    //---------------------------------------------------------------------
    // 6. RESET CHANNEL STATUS
    //---------------------------------------------------------------------
    ChannelStatus.Enable := FALSE;
    ChannelStatus.Online := FALSE;
    ChannelStatus.Ready := FALSE;
    ChannelStatus.Busy := FALSE;
    ChannelStatus.ResultReady := FALSE;
    ChannelStatus.Error := FALSE;
    ChannelStatus.CurrentJobID := 0;
    ChannelStatus.CurrentTriggerID := 0;
    ChannelStatus.ResultStatus := E_VisionResultStatus.VIS_RESULT_NONE;

    tHeartbeatTimeout(IN := FALSE);

    RETURN;
END_IF;


//=============================================================================
// DISABLE
//=============================================================================
IF NOT Enable THEN

    Registers[uiR2V + 0] := WORD#0;

    Active := FALSE;
    Error := FALSE;
    ErrorID := 0;

    ChannelStatus.Enable := FALSE;
    ChannelStatus.Online := FALSE;
    ChannelStatus.Ready := FALSE;
    ChannelStatus.Busy := FALSE;
    ChannelStatus.ResultReady := FALSE;
    ChannelStatus.Error := FALSE;

    RETURN;
END_IF;


//=============================================================================
// NORMAL RUN
//=============================================================================
Active := TRUE;
ChannelStatus.Enable := TRUE;

// Active := TRUE;
// ChannelStatus.Enable := TRUE;

// //=============================================================================
// // MEMORY BASE / SCALE
// //=============================================================================
// uiBase := Config.BaseAddress;
// uiR2V := uiBase + Config.CommandOffset;
// uiV2R := uiBase + Config.StatusOffset;
// uiData := uiBase + Config.DataOffset;
// uiMulti := uiBase + 132;                            // MultiData cố định theo mapping V1.1.
// 
// IF uiR2V + 99 > 1199 OR uiV2R + 199 > 1199 THEN
//     Error := TRUE;
//     ErrorID := 9251;                                // Base/Offset vượt vùng MODBUS.
//     RETURN;
// END_IF;

Error := FALSE;
ErrorID := 0;
rPositionScale := Config.PositionScale;
rAngleScale := Config.AngleScale;
rScoreScale := Config.ScoreScale;
IF ABS(rPositionScale) <= GVL.C_EPSILON THEN rPositionScale := 1.0; END_IF;
IF ABS(rAngleScale) <= GVL.C_EPSILON THEN rAngleScale := 1.0; END_IF;
IF ABS(rScoreScale) <= GVL.C_EPSILON THEN rScoreScale := 1.0; END_IF;

//=============================================================================
// 1. ROBOT -> VISION: CONTROL WORD + COMMAND
//=============================================================================
// Heartbeat dùng biến nội bộ toggle; KHÔNG đảo trực tiếp register mỗi scan Communication.
xHeartbeatToggle := NOT xHeartbeatToggle;

wControl := WORD#0;
wControl.0 := xHeartbeatToggle;
wControl.1 := Command.Execute;
wControl.2 := ModbusControl.RunCalib;
wControl.3 := ModbusControl.CalibPosReady;
wControl.4 := ModbusControl.AckResult;
wControl.5 := ModbusControl.AckBlock;
wControl.6 := Command.Reset;
wControl.7 := Command.Abort;
Registers[uiR2V + 0] := wControl;
Registers[uiR2V + 1] := UINT_TO_WORD(Command.JobID);

CASE Command.Application OF
    E_VisionApplication.VIS_APP_ALIGN: Registers[uiR2V + 2] := WORD#10;
    E_VisionApplication.VIS_APP_INSPECTION: Registers[uiR2V + 2] := WORD#20;
    E_VisionApplication.VIS_APP_SINGLE_POINT: Registers[uiR2V + 2] := WORD#30;
    E_VisionApplication.VIS_APP_POINT_LIST: Registers[uiR2V + 2] := WORD#40;
    E_VisionApplication.VIS_APP_GLUE_PATH: Registers[uiR2V + 2] := WORD#50;
    E_VisionApplication.VIS_APP_PICK_POSITION: Registers[uiR2V + 2] := WORD#60;
    E_VisionApplication.VIS_APP_CONVEYOR_PICK: Registers[uiR2V + 2] := WORD#70;
    E_VisionApplication.VIS_APP_CONVEYOR_INSPECTION: Registers[uiR2V + 2] := WORD#80;
    E_VisionApplication.VIS_APP_CONVEYOR_GLUE: Registers[uiR2V + 2] := WORD#90;
    E_VisionApplication.VIS_APP_CALIBRATION: Registers[uiR2V + 2] := WORD#100;
    ELSE Registers[uiR2V + 2] := WORD#0;
END_CASE;

Registers[uiR2V + 3] := F_VisionUDINTLowWord(Command.TriggerID);
Registers[uiR2V + 4] := F_VisionUDINTHighWord(Command.TriggerID);
Registers[uiR2V + 5] := UINT_TO_WORD(ModbusControl.CalibPointCount);
Registers[uiR2V + 6] := UINT_TO_WORD(ModbusControl.RequestBlockIndex);
Registers[uiR2V + 7] := UINT_TO_WORD(ModbusControl.AckBlockIndex);
Registers[uiR2V + 8] := UINT_TO_WORD(ModbusControl.CommandCode);
Registers[uiR2V + 9] := WORD#0;

// 12 Calibration Point; mỗi Point = X/Y/A, mỗi thành phần = LOW/HIGH WORD.
FOR uiPoint := 1 TO 12 DO
    diRaw := F_VisionRealToRawDINT(ModbusControl.CalibrationPoints[uiPoint].X, rPositionScale);
    Registers[uiR2V + 10 + (uiPoint - 1) * 6] := F_VisionDINTLowWord(diRaw);
    Registers[uiR2V + 11 + (uiPoint - 1) * 6] := F_VisionDINTHighWord(diRaw);

    diRaw := F_VisionRealToRawDINT(ModbusControl.CalibrationPoints[uiPoint].Y, rPositionScale);
    Registers[uiR2V + 12 + (uiPoint - 1) * 6] := F_VisionDINTLowWord(diRaw);
    Registers[uiR2V + 13 + (uiPoint - 1) * 6] := F_VisionDINTHighWord(diRaw);

    diRaw := F_VisionRealToRawDINT(ModbusControl.CalibrationPoints[uiPoint].A, rAngleScale);
    Registers[uiR2V + 14 + (uiPoint - 1) * 6] := F_VisionDINTLowWord(diRaw);
    Registers[uiR2V + 15 + (uiPoint - 1) * 6] := F_VisionDINTHighWord(diRaw);
END_FOR;

// Capture reference của command runtime.
diRaw := F_VisionRealToRawDINT(Command.CaptureConveyorPos, rPositionScale);
Registers[uiR2V + 82] := F_VisionDINTLowWord(diRaw);
Registers[uiR2V + 83] := F_VisionDINTHighWord(diRaw);

diRaw := F_VisionRealToRawDINT(Command.CaptureRobotPos.X, rPositionScale);
Registers[uiR2V + 84] := F_VisionDINTLowWord(diRaw);
Registers[uiR2V + 85] := F_VisionDINTHighWord(diRaw);

diRaw := F_VisionRealToRawDINT(Command.CaptureRobotPos.Y, rPositionScale);
Registers[uiR2V + 86] := F_VisionDINTLowWord(diRaw);
Registers[uiR2V + 87] := F_VisionDINTHighWord(diRaw);

diRaw := F_VisionRealToRawDINT(Command.CaptureRobotPos.A, rAngleScale);
Registers[uiR2V + 88] := F_VisionDINTLowWord(diRaw);
Registers[uiR2V + 89] := F_VisionDINTHighWord(diRaw);

//=============================================================================
// 2. VISION -> ROBOT: STATUS WORD
//=============================================================================
wStatus := Registers[uiV2R + 0];
ModbusStatus.HeartBeat := wStatus.0;
ModbusStatus.TriggerDone := wStatus.1;
ModbusStatus.CalibDone := wStatus.2;
ModbusStatus.ResultReady := wStatus.3;
ModbusStatus.Busy := wStatus.4;
ModbusStatus.Run1Slot := wStatus.5;
ModbusStatus.BlockReady := wStatus.6;
ModbusStatus.Error := wStatus.7;
ModbusStatus.CalibBusy := wStatus.8;
ModbusStatus.CalibError := wStatus.9;

ChannelStatus.Ready := NOT ModbusStatus.Busy AND NOT ModbusStatus.Error;
ChannelStatus.Busy := ModbusStatus.Busy;
ChannelStatus.ResultReady := ModbusStatus.ResultReady;
ChannelStatus.Error := ModbusStatus.Error;

// Heartbeat timeout 2 s: mỗi lần bit đổi thì reset timer.
IF ModbusStatus.HeartBeat <> xLastHeartbeat THEN
    xLastHeartbeat := ModbusStatus.HeartBeat;
    ChannelStatus.Online := TRUE;
    tHeartbeatTimeout(IN := FALSE);
ELSE
    tHeartbeatTimeout(IN := TRUE, PT := T#2S);
    IF tHeartbeatTimeout.Q THEN ChannelStatus.Online := FALSE; END_IF;
END_IF;

//=============================================================================
// 3. RESULT HEADER
//=============================================================================
ChannelStatus.CurrentJobID := WORD_TO_UINT(Registers[uiV2R + 1]);
udiTriggerID := F_VisionWordsToUDINT_LH(Registers[uiV2R + 4], Registers[uiV2R + 5]);
ChannelStatus.CurrentTriggerID := udiTriggerID;

VisionResult.Header.CameraID := Config.CameraID;
VisionResult.Header.JobID := WORD_TO_UINT(Registers[uiV2R + 1]);
VisionResult.Header.TriggerID := udiTriggerID;
VisionResult.Header.ResultCode := WORD_TO_UINT(Registers[uiV2R + 7]);
VisionResult.Header.ErrorCode := WORD_TO_UINT(Registers[uiV2R + 7]);
VisionResult.Header.DataCount := WORD_TO_UINT(Registers[uiV2R + 8]);
VisionResult.Header.BlockCount := WORD_TO_UINT(Registers[uiV2R + 9]);
VisionResult.Header.BlockIndex := WORD_TO_UINT(Registers[uiV2R + 10]);
VisionResult.Header.BlockDataCount := WORD_TO_UINT(Registers[uiV2R + 11]);
VisionResult.Header.Checksum := F_VisionWordsToUDINT_LH(Registers[uiV2R + 12], Registers[uiV2R + 13]);

diRaw := F_VisionWordsToDINT_LH(Registers[uiV2R + 14], Registers[uiV2R + 15]);
VisionResult.Header.CaptureConveyorPos := DINT_TO_REAL(diRaw) * rPositionScale;
ModbusStatus.BlockIndex := VisionResult.Header.BlockIndex;
ModbusStatus.BlockDataCount := VisionResult.Header.BlockDataCount;

CASE WORD_TO_UINT(Registers[uiV2R + 2]) OF
    10: VisionResult.Header.Application := E_VisionApplication.VIS_APP_ALIGN;
    20: VisionResult.Header.Application := E_VisionApplication.VIS_APP_INSPECTION;
    30: VisionResult.Header.Application := E_VisionApplication.VIS_APP_SINGLE_POINT;
    40: VisionResult.Header.Application := E_VisionApplication.VIS_APP_POINT_LIST;
    50: VisionResult.Header.Application := E_VisionApplication.VIS_APP_GLUE_PATH;
    60: VisionResult.Header.Application := E_VisionApplication.VIS_APP_PICK_POSITION;
    70: VisionResult.Header.Application := E_VisionApplication.VIS_APP_CONVEYOR_PICK;
    80: VisionResult.Header.Application := E_VisionApplication.VIS_APP_CONVEYOR_INSPECTION;
    90: VisionResult.Header.Application := E_VisionApplication.VIS_APP_CONVEYOR_GLUE;
    100: VisionResult.Header.Application := E_VisionApplication.VIS_APP_CALIBRATION;
    ELSE VisionResult.Header.Application := E_VisionApplication.VIS_APP_NONE;
END_CASE;

CASE WORD_TO_UINT(Registers[uiV2R + 3]) OF
    10: VisionResult.Header.DataType := E_VisionDataType.VIS_DATA_BOOL;
    20: VisionResult.Header.DataType := E_VisionDataType.VIS_DATA_VALUE;
    30: VisionResult.Header.DataType := E_VisionDataType.VIS_DATA_POS;
    40: VisionResult.Header.DataType := E_VisionDataType.VIS_DATA_ALIGN;
    50: VisionResult.Header.DataType := E_VisionDataType.VIS_DATA_INSPECTION;
    60: VisionResult.Header.DataType := E_VisionDataType.VIS_DATA_POINT_LIST;
    70: VisionResult.Header.DataType := E_VisionDataType.VIS_DATA_GLUE_PATH;
    80: VisionResult.Header.DataType := E_VisionDataType.VIS_DATA_TRACK_OBJECT;
    ELSE VisionResult.Header.DataType := E_VisionDataType.VIS_DATA_NONE;
END_CASE;

CASE WORD_TO_UINT(Registers[uiV2R + 6]) OF
    10: VisionResult.Header.ResultStatus := E_VisionResultStatus.VIS_RESULT_PENDING;
    20: VisionResult.Header.ResultStatus := E_VisionResultStatus.VIS_RESULT_OK;
    30: VisionResult.Header.ResultStatus := E_VisionResultStatus.VIS_RESULT_NG;
    40: VisionResult.Header.ResultStatus := E_VisionResultStatus.VIS_RESULT_NOT_FOUND;
    50: VisionResult.Header.ResultStatus := E_VisionResultStatus.VIS_RESULT_LOW_SCORE;
    60: VisionResult.Header.ResultStatus := E_VisionResultStatus.VIS_RESULT_OUT_OF_RANGE;
    70: VisionResult.Header.ResultStatus := E_VisionResultStatus.VIS_RESULT_INCOMPLETE;
    80: VisionResult.Header.ResultStatus := E_VisionResultStatus.VIS_RESULT_INVALID;
    900: VisionResult.Header.ResultStatus := E_VisionResultStatus.VIS_RESULT_ERROR;
    ELSE VisionResult.Header.ResultStatus := E_VisionResultStatus.VIS_RESULT_NONE;
END_CASE;
ChannelStatus.ResultStatus := VisionResult.Header.ResultStatus;

// Vision đã hạ ResultReady: kết thúc handshake Result trước.
IF NOT ModbusStatus.ResultReady THEN
    ModbusControl.AckResult := FALSE;
    ModbusControl.AckBlock := FALSE;
    ModbusControl.AckBlockIndex := 0;
    ModbusControl.RequestBlockIndex := 0;
END_IF;

//=============================================================================
// 4. SIMPLE RESULT - POS / ALIGN
//=============================================================================
IF ModbusStatus.ResultReady AND udiTriggerID <> 0 AND udiTriggerID <> udiLastResultTriggerID
AND (VisionResult.Header.DataType = E_VisionDataType.VIS_DATA_POS OR VisionResult.Header.DataType = E_VisionDataType.VIS_DATA_ALIGN) THEN

    diRaw := F_VisionWordsToDINT_LH(Registers[uiData + 0], Registers[uiData + 1]);
    VisionResult.PosResult.Pos.X := DINT_TO_REAL(diRaw) * rPositionScale;
    diRaw := F_VisionWordsToDINT_LH(Registers[uiData + 2], Registers[uiData + 3]);
    VisionResult.PosResult.Pos.Y := DINT_TO_REAL(diRaw) * rPositionScale;
    diRaw := F_VisionWordsToDINT_LH(Registers[uiData + 4], Registers[uiData + 5]);
    VisionResult.PosResult.Pos.A := DINT_TO_REAL(diRaw) * rAngleScale;

    VisionResult.PosResult.Pos.Z := 0.0;
    VisionResult.PosResult.Score := UINT_TO_REAL(WORD_TO_UINT(Registers[uiData + 6])) * rScoreScale;
    VisionResult.PosResult.Valid := Registers[uiData + 7].0;
    VisionResult.PosResult.FeatureID := WORD_TO_UINT(Registers[uiData + 8]);

    IF VisionResult.Header.DataType = E_VisionDataType.VIS_DATA_ALIGN THEN
        VisionResult.AlignResult.Valid := VisionResult.PosResult.Valid;
        VisionResult.AlignResult.RawOffset := VisionResult.PosResult.Pos;
        VisionResult.AlignResult.RobotOffset := VisionResult.PosResult.Pos;
        VisionResult.AlignResult.Score := VisionResult.PosResult.Score;
        VisionResult.AlignResult.FeatureID := VisionResult.PosResult.FeatureID;
    END_IF;

    VisionResult.Header.Valid := TRUE;
    udiLastResultTriggerID := udiTriggerID;
    ModbusControl.AckResult := TRUE;
END_IF;

//=============================================================================
// 5. TRACKING MULTI-BLOCK
//=============================================================================
IF ModbusStatus.ResultReady AND ModbusStatus.BlockReady
AND VisionResult.Header.DataType = E_VisionDataType.VIS_DATA_TRACK_OBJECT THEN

    uiBlockIndex := VisionResult.Header.BlockIndex;
    uiBlockDataCount := VisionResult.Header.BlockDataCount;

    IF uiBlockIndex = 0 OR uiBlockIndex > VisionResult.Header.BlockCount THEN
        Error := TRUE;
        ErrorID := 9252;
    ELSIF uiBlockDataCount > 10 THEN
        Error := TRUE;
        ErrorID := 9253;
    ELSIF udiTriggerID <> udiLastBlockTriggerID OR uiBlockIndex <> uiLastDecodedBlock THEN

        // Block đầu của Trigger mới: xóa Result cũ trước khi ghép frame mới.
        IF uiBlockIndex = 1 THEN
            VisionResult.Header.Valid := FALSE;
            VisionResult.TrackObjectResult.Valid := FALSE;
            VisionResult.TrackObjectResult.ObjectCount := 0;
            FOR uiRecord := 1 TO GVL.C_MAX_VISION_TRACK_OBJECTS_PER_FRAME DO
                VisionResult.TrackObjectResult.Objects[uiRecord].Valid := FALSE;
            END_FOR;
        END_IF;

        FOR uiRecord := 1 TO uiBlockDataCount DO
            uiGlobalObject := (uiBlockIndex - 1) * 10 + uiRecord;

            IF uiGlobalObject <= GVL.C_MAX_VISION_TRACK_OBJECTS_PER_FRAME THEN
                wObjectInfo := Registers[uiMulti + (uiRecord - 1) * 9 + 6];

                diRaw := F_VisionWordsToDINT_LH(Registers[uiMulti + (uiRecord - 1) * 9 + 0], Registers[uiMulti + (uiRecord - 1) * 9 + 1]);
                VisionResult.TrackObjectResult.Objects[uiGlobalObject].Pos.X := DINT_TO_REAL(diRaw) * rPositionScale;

                diRaw := F_VisionWordsToDINT_LH(Registers[uiMulti + (uiRecord - 1) * 9 + 2], Registers[uiMulti + (uiRecord - 1) * 9 + 3]);
                VisionResult.TrackObjectResult.Objects[uiGlobalObject].Pos.Y := DINT_TO_REAL(diRaw) * rPositionScale;

                diRaw := F_VisionWordsToDINT_LH(Registers[uiMulti + (uiRecord - 1) * 9 + 4], Registers[uiMulti + (uiRecord - 1) * 9 + 5]);
                VisionResult.TrackObjectResult.Objects[uiGlobalObject].Pos.A := DINT_TO_REAL(diRaw) * rAngleScale;

                VisionResult.TrackObjectResult.Objects[uiGlobalObject].Pos.Z := 0.0;
                VisionResult.TrackObjectResult.Objects[uiGlobalObject].Valid := wObjectInfo.0;
                VisionResult.TrackObjectResult.Objects[uiGlobalObject].Score := UINT_TO_REAL(WORD_TO_UINT(Registers[uiMulti + (uiRecord - 1) * 9 + 7])) * rScoreScale;
                VisionResult.TrackObjectResult.Objects[uiGlobalObject].ProductClassID := WORD_TO_UINT(Registers[uiMulti + (uiRecord - 1) * 9 + 8]);
                VisionResult.TrackObjectResult.Objects[uiGlobalObject].FeatureID := 0; // V1.1 không truyền FeatureID.
            END_IF;
        END_FOR;

        udiLastBlockTriggerID := udiTriggerID;
        uiLastDecodedBlock := uiBlockIndex;
        ModbusControl.AckBlock := TRUE;
        ModbusControl.AckBlockIndex := uiBlockIndex;

        IF uiBlockIndex < VisionResult.Header.BlockCount THEN
            ModbusControl.RequestBlockIndex := uiBlockIndex + 1;
        ELSE
            VisionResult.TrackObjectResult.ObjectCount := VisionResult.Header.DataCount;
            IF VisionResult.TrackObjectResult.ObjectCount > GVL.C_MAX_VISION_TRACK_OBJECTS_PER_FRAME THEN
                VisionResult.TrackObjectResult.ObjectCount := GVL.C_MAX_VISION_TRACK_OBJECTS_PER_FRAME;
            END_IF;

            VisionResult.TrackObjectResult.Valid := TRUE;
            VisionResult.Header.Valid := TRUE;
            udiLastResultTriggerID := udiTriggerID;
            ModbusControl.RequestBlockIndex := 0;
            ModbusControl.AckResult := TRUE;
        END_IF;
    END_IF;
ELSE
    // Khi PC hạ/chuyển BlockReady thì PLC hạ AckBlock để handshake Block kế tiếp.
    ModbusControl.AckBlock := FALSE;
END_IF;

END_FUNCTION_BLOCK

// Just_Motion_Control_x86_64_Linux_SM_WV/Application/FC_/Vision/F_VisionUDINTLowWord
FUNCTION F_VisionUDINTLowWord : WORD
VAR_INPUT Value : UDINT; END_VAR

F_VisionUDINTLowWord := DWORD_TO_WORD(UDINT_TO_DWORD(Value) AND DWORD#16#0000FFFF);

END_FUNCTION

// Just_Motion_Control_x86_64_Linux_SM_WV/Application/FC_/Vision/F_VisionUDINTHighWord
FUNCTION F_VisionUDINTHighWord : WORD
VAR_INPUT Value : UDINT; END_VAR

F_VisionUDINTHighWord := DWORD_TO_WORD(SHR(UDINT_TO_DWORD(Value), 16));

END_FUNCTION

// Just_Motion_Control_x86_64_Linux_SM_WV/Application/FC_/Vision/F_VisionRealToRawDINT
FUNCTION F_VisionRealToRawDINT : DINT
VAR_INPUT
    Value : REAL;
    Scale : REAL;
END_VAR

IF ABS(Scale) <= GVL.C_REAL_EPSILON THEN
    F_VisionRealToRawDINT := 0;
ELSE
    F_VisionRealToRawDINT := REAL_TO_DINT(Value / Scale);
END_IF;

END_FUNCTION

// Just_Motion_Control_x86_64_Linux_SM_WV/Application/FC_/Vision/F_VisionDINTLowWord
FUNCTION F_VisionDINTLowWord : WORD
VAR_INPUT Value : DINT; END_VAR
VAR dwValue : DWORD; END_VAR

dwValue := DINT_TO_DWORD(Value);
F_VisionDINTLowWord := DWORD_TO_WORD(dwValue AND DWORD#16#0000FFFF);

END_FUNCTION

// Just_Motion_Control_x86_64_Linux_SM_WV/Application/FC_/Vision/F_VisionDINTHighWord
FUNCTION F_VisionDINTHighWord : WORD
VAR_INPUT Value : DINT; END_VAR
VAR dwValue : DWORD; END_VAR

dwValue := DINT_TO_DWORD(Value);
F_VisionDINTHighWord := DWORD_TO_WORD(SHR(dwValue, 16));

END_FUNCTION

// Just_Motion_Control_x86_64_Linux_SM_WV/Application/FC_/Vision/F_VisionWordsToUDINT_LH
FUNCTION F_VisionWordsToUDINT_LH : UDINT
VAR_INPUT
    LowWord : WORD;
    HighWord : WORD;
END_VAR
VAR
    dwValue : DWORD;
END_VAR

dwValue := SHL(WORD_TO_DWORD(HighWord), 16) OR WORD_TO_DWORD(LowWord);
F_VisionWordsToUDINT_LH := DWORD_TO_UDINT(dwValue);

END_FUNCTION

// Just_Motion_Control_x86_64_Linux_SM_WV/Application/FC_/Vision/F_VisionWordsToDINT_LH
FUNCTION F_VisionWordsToDINT_LH : DINT
VAR_INPUT
    LowWord : WORD;
    HighWord : WORD;
END_VAR
VAR
    dwValue : DWORD;
END_VAR

dwValue := SHL(WORD_TO_DWORD(HighWord), 16) OR WORD_TO_DWORD(LowWord);
F_VisionWordsToDINT_LH := DWORD_TO_DINT(dwValue);

END_FUNCTION

// Just_Motion_Control_x86_64_Linux_SM_WV/Application/FB_/FB_MotionQueuePush
FUNCTION_BLOCK FB_MotionQueuePush
VAR_INPUT
	Item : ST_MotionQueueItem;
    Execute : BOOL;
END_VAR
VAR_OUTPUT
	Done : BOOL;
    Error : BOOL;
	Busy  : BOOL;
END_VAR
VAR
	ExecuteOld  : BOOL;
	ExecuteRise : BOOL;
END_VAR

// ExecuteRise := Execute AND NOT ExecuteOld; // Tao xung canh len 
// ExecuteOld := Execute;
// 
// Done := FALSE;
// Error := FALSE;
// 
// IF ExecuteRise THEN
//     IF GVL.A_MotionCount >= 20 THEN // Kiểm tra Queue đầy chưa
//         Error := TRUE;
//     ELSE
//         GVL.A_MotionQueue[GVL.A_MotionTail] := Item; // Ghi du lieu vao Queue
// 
//         GVL.A_MotionTail := GVL.A_MotionTail + 1; // Dich vi tri ghi du lieu
//         IF GVL.A_MotionTail > 20 THEN  // Queue vong tron
//             GVL.A_MotionTail := 1;
//         END_IF;
// 
//         GVL.A_MotionCount := GVL.A_MotionCount + 1; // Tang so luong Item trong Queue
//         Done := TRUE;  //Push thanh cong
//     END_IF;
// END_IF;

//====================================================
// FB_MotionQueuePush
// Execute = TRUE  -> Push đúng 1 lần
// Done/Error giữ đến khi Execute = FALSE
//====================================================

IF NOT Execute THEN

    Done := FALSE;
    Error := FALSE;
    Busy := FALSE;

ELSE

    IF NOT Busy THEN

        Busy := TRUE;

        IF GVL.A_MotionCount >= 20 THEN

            Error := TRUE;
            Done := FALSE;

        ELSE

            GVL.A_MotionQueue[GVL.A_MotionTail] := Item;

            GVL.A_MotionTail := GVL.A_MotionTail + 1;

            IF GVL.A_MotionTail > 20 THEN
                GVL.A_MotionTail := 1;
            END_IF;

            GVL.A_MotionCount := GVL.A_MotionCount + 1;

            Done := TRUE;
            Error := FALSE;

        END_IF;

    END_IF;

END_IF;

END_FUNCTION_BLOCK

// Just_Motion_Control_x86_64_Linux_SM_WV/Application/FB_/FB_MotionQueuePop
FUNCTION_BLOCK FB_MotionQueuePop
VAR_INPUT
	Execute : BOOL;
END_VAR
VAR_OUTPUT
	Item  : ST_MotionQueueItem;
    Done  : BOOL;
    Empty : BOOL;
	Busy  : BOOL;
END_VAR
VAR
	ExecuteOld  : BOOL;
	ExecuteRise : BOOL;
END_VAR

// ExecuteRise := Execute AND NOT ExecuteOld; // Tao xung suon len
// ExecuteOld := Execute;
// 
// Done := FALSE;
// Empty := FALSE;
// 
// IF ExecuteRise THEN // Chỉ xử lý khi có lệnh gọi pop
//     IF GVL.A_MotionCount <= 0 THEN // Nếu số phần tử trong queue bằng 0 hoặc nhỏ hơn 0 thì queue rỗng
//         Empty := TRUE;
//     ELSE
//         Item := GVL.A_MotionQueue[GVL.A_MotionHead];  // Nếu queue còn dữ liệu thì lấy phần tử tại vị trí A_MotionHead
// 
//         GVL.A_MotionHead := GVL.A_MotionHead + 1; // Tang gia tri len 1 sau khi lay
//         IF GVL.A_MotionHead > 20 THEN // Nếu Head vượt quá 20 thì quay lại 1
//             GVL.A_MotionHead := 1;
//         END_IF;
// 
//         GVL.A_MotionCount := GVL.A_MotionCount - 1; // giam so luong phan di trong queue di 1
//         Done := TRUE;
//     END_IF;
// END_IF;

//====================================================
// FB_MotionQueuePop
// Handshake:
// Execute = TRUE  -> xử lý đúng 1 lần
// Done/Empty giữ TRUE cho tới khi Execute = FALSE
//====================================================

IF NOT Execute THEN

    Done := FALSE;
    Empty := FALSE;
    Busy := FALSE;

ELSE

    IF NOT Busy THEN

        Busy := TRUE;

        IF GVL.A_MotionCount <= 0 THEN

            Empty := TRUE;
            Done := FALSE;

        ELSE

            Item := GVL.A_MotionQueue[GVL.A_MotionHead];

            GVL.A_MotionHead := GVL.A_MotionHead + 1; // Tang gia tri len 1 sau khi lay

            IF GVL.A_MotionHead > 20 THEN // Nếu Head vượt quá 20 thì quay lại 1
                GVL.A_MotionHead := 1;
            END_IF;

            GVL.A_MotionCount := GVL.A_MotionCount - 1; // giam so luong phan di trong queue di 1

            Done := TRUE;
            Empty := FALSE;

        END_IF;

    END_IF;

END_IF;

END_FUNCTION_BLOCK

// Just_Motion_Control_x86_64_Linux_SM_WV/Application/FB_/FB_RunMoveP
FUNCTION_BLOCK FB_RunMoveP
VAR_INPUT
    Start       : BOOL;
    Item        : ST_MotionQueueItem;
    PositionIn  : SMC_POS_REF;
    CoordSystem : SMC_COORD_SYSTEM;
    AcceptTimeoutTime : TIME := T#2S;
    MoveTimeoutTime   : TIME := T#100S;
    PosCheckDelayTime : TIME := T#13MS;
END_VAR
VAR_IN_OUT
	AxisGroup   : AXIS_GROUP_REF_SM3;
	Release : BOOL;
END_VAR
VAR_OUTPUT
    Accepted       : BOOL;
    Done           : BOOL;
    Busy           : BOOL;
    Active         : BOOL;
    Error          : BOOL;
    Timeout        : BOOL;
    Aborted        : BOOL;
    ErrorID        : SMC_ERROR;
    ErrorID_Custom : INT;
    State          : E_MoveState;
END_VAR

VAR
    fbMoveP : MC_MoveDirectAbsolute;

    tAcceptTimeout : TON;
    tMoveTimeout   : TON;
    tPosCheckDelay : TON;

    StartEdge    : BOOL;
    LastStart    : BOOL;
    ExecutePulse : BOOL;

    PosBuf : SMC_POS_REF;
	DonePosition : SM3_Robotics.SMC_POS_REF;
    BufferMode : SM3_Robotics.MC_BUFFER_MODE;
    TransMode  : SM3_Robotics.MC_TRANSITION_MODE;
    TransParam : ARRAY[0..(SMC_RCNST.MAX_TRANS_PARAMS - 1)] OF LREAL := [0.0, 0.0];

    VelFacLocal    : LREAL;
    AccFacLocal    : LREAL;
    JerkFacLocal   : LREAL;
    TorqueFacLocal : LREAL;
END_VAR

VAR CONSTANT
    C_BM_Buffered     : SM3_Robotics.MC_BUFFER_MODE := 1;
    C_BM_BlendingNext : SM3_Robotics.MC_BUFFER_MODE := 4;

    C_TM_CornerDistance : SM3_Robotics.MC_TRANSITION_MODE := 2;
    C_TM_None           : SM3_Robotics.MC_TRANSITION_MODE := 0;
    C_TM_StartVelocity  : SM3_Robotics.MC_TRANSITION_MODE := 1;
END_VAR

//============================================================
// FB_RunMoveP
// Mục tiêu kiểm nghiệm:
// - Execute được giữ đến khi SoftMotion nhận lệnh.
// - Accepted được latch, không bị mất xung.
// - Done được giữ đến khi MotionManager hạ Start.
//============================================================

//------------------------------------------------------------
// Phát hiện cạnh lên Start
//------------------------------------------------------------
StartEdge := Start AND NOT LastStart;
LastStart := Start;


//------------------------------------------------------------
// Giá trị mặc định của Execute
// Execute sẽ được bật trong MOVE_SEND và MOVE_WAIT_ACCEPT
//------------------------------------------------------------
ExecutePulse := FALSE;


//============================================================
// STATE MACHINE
//============================================================
CASE State OF

	//========================================================
	// IDLE
	//========================================================
	E_MoveState.MOVE_IDLE:

		// Output trạng thái
		Accepted := FALSE;
		Done := FALSE;
		Error := FALSE;
		Timeout := FALSE;
		Aborted := FALSE;
		Release := FALSE;
 
		ErrorID_Custom := 0;

		// Reset timer
		tAcceptTimeout(IN := FALSE);
		tMoveTimeout(IN := FALSE);
		tPosCheckDelay(IN := FALSE);

//         IF StartEdge THEN
		IF Start AND NOT fbMoveP.Busy AND NOT fbMoveP.Active THEN	
			//------------------------------------------------
			// Chốt tọa độ tại thời điểm bắt đầu
			//------------------------------------------------
			PosBuf := PositionIn;

			//------------------------------------------------
			// MoveP dùng các hệ số Factor
			//------------------------------------------------
			
			IF AxisGroup.m_id = SCARA_A.m_id THEN
				VelFacLocal    := GVL_1.DATA_RB_A.Fac_Vel;
				AccFacLocal    := GVL_1.DATA_RB_A.Fac_Acc;
				JerkFacLocal   := GVL_1.DATA_RB_A.Fac_Jerk;
				TorqueFacLocal := GVL_1.DATA_RB_A.Fac_Torque;
			ELSE
				VelFacLocal    := GVL_1.DATA_RB_B.Fac_Vel;
				AccFacLocal    := GVL_1.DATA_RB_B.Fac_Acc;
				JerkFacLocal   := GVL_1.DATA_RB_B.Fac_Jerk;
				TorqueFacLocal := GVL_1.DATA_RB_B.Fac_Torque;
			END_IF

			//------------------------------------------------
			// Giá trị dự phòng an toàn
			//------------------------------------------------
			IF VelFacLocal <= 0.0 THEN
				VelFacLocal := 0.1;
			END_IF;

			IF AccFacLocal <= 0.0 THEN
				AccFacLocal := 0.1;
			END_IF;

			IF JerkFacLocal <= 0.0 THEN
				JerkFacLocal := 0.1;
			END_IF;

			IF TorqueFacLocal <= 0.0 THEN
				TorqueFacLocal := 0.1;
			END_IF;

			//------------------------------------------------
			// Mapping Blend
			//------------------------------------------------
			IF (Item.BlendMode = 0)
			   OR (Item.BlendRadius <= 0.0)
			THEN
				// Không blend
				BufferMode := C_BM_Buffered;
				TransMode := C_TM_None;

				TransParam[0] := 0.0;
				TransParam[1] := 0.0;

			ELSE
				// Có blend
				//BufferMode := C_BM_BlendingNext;
				BufferMode := GVL.C_BM_BlendingHigh;

				CASE Item.BlendMode OF

					1:
						TransMode := C_TM_CornerDistance;

					2:
						TransMode := C_TM_StartVelocity;

				ELSE
					TransMode := C_TM_CornerDistance;

				END_CASE;

				TransParam[0] := Item.BlendRadius;
				TransParam[1] := 0.0;
			END_IF;

			//------------------------------------------------
			// Reset output cho lệnh mới
			//------------------------------------------------
			Accepted := FALSE;
			Done := FALSE;
			Error := FALSE;
			Timeout := FALSE;
			Aborted := FALSE;
			ErrorID_Custom := 0;

			//------------------------------------------------
			// Chuyển sang gửi lệnh
			//------------------------------------------------
			State := E_MoveState.MOVE_SEND;

		END_IF;


	//========================================================
	// SEND COMMAND
	//========================================================
	E_MoveState.MOVE_SEND:

		// Giữ Execute TRUE
		ExecutePulse := TRUE;

		// Bắt đầu timeout nhận lệnh
		tAcceptTimeout(
			IN := TRUE,
			PT := AcceptTimeoutTime
		);

		State := E_MoveState.MOVE_WAIT_ACCEPT;


	//========================================================
	// WAIT COMMAND ACCEPTED
	//========================================================
	E_MoveState.MOVE_WAIT_ACCEPT:

		//--------------------------------------------------------
	// Giữ Execute TRUE cho đến khi SoftMotion xác nhận
	// đã nhận đúng lệnh mới
	//--------------------------------------------------------
	ExecutePulse := TRUE;

	tAcceptTimeout(
		IN := TRUE,
		PT := AcceptTimeoutTime
	);

	//--------------------------------------------------------
	// Chỉ CommandAccepted mới được coi là Accepted.
	// Không dùng Busy/Active vì có thể là trạng thái còn lại
	// của chuyển động trước.
	//--------------------------------------------------------
	IF fbMoveP.CommandAccepted THEN

		Accepted := TRUE;
		ExecutePulse := FALSE;

		tAcceptTimeout(IN := FALSE);

		tMoveTimeout(
			IN := TRUE,
			PT := MoveTimeoutTime
		);

		State := E_MoveState.MOVE_WAIT_DONE;

	ELSIF fbMoveP.CommandAborted THEN

		ExecutePulse := FALSE;

		Aborted := TRUE;
		Error := TRUE;
		ErrorID_Custom := 5003;

		tAcceptTimeout(IN := FALSE);
		State := E_MoveState.MOVE_ABORTED;

	ELSIF fbMoveP.Error THEN

		ExecutePulse := FALSE;

		Error := TRUE;
		ErrorID := fbMoveP.ErrorID;
		ErrorID_Custom := 5004;

		tAcceptTimeout(IN := FALSE);
		State := E_MoveState.MOVE_ERROR;

	ELSIF tAcceptTimeout.Q THEN

		ExecutePulse := FALSE;

		Timeout := TRUE;
		Error := TRUE;
		ErrorID_Custom := 5005;

		tAcceptTimeout(IN := FALSE);
		State := E_MoveState.MOVE_TIMEOUT;

	END_IF;


	//========================================================
	// WAIT MOTION DONE
	//========================================================
	E_MoveState.MOVE_WAIT_DONE:

		// Giữ Accepted để MotionManager chắc chắn đọc được
		Accepted := TRUE;

		ExecutePulse := FALSE;

		tMoveTimeout(
			IN := TRUE,
			PT := MoveTimeoutTime
		);

		IF fbMoveP.Done THEN

			tMoveTimeout(IN := FALSE);
			//DonePosition := POU_MONITOR_ROBOT.RB1_POS;
			//------------------------------------------------
			// Không blend: kiểm tra vị trí cuối
			//------------------------------------------------
			//IF ((Item.BlendMode = 0) OR (Item.BlendRadius <= 0.0)) AND (NOT Item.SkipPositionCheck) THEN
			IF (NOT Item.SkipPositionCheck) THEN
				tPosCheckDelay(
					IN := TRUE,
					PT := PosCheckDelayTime
				);

				State := E_MoveState.MOVE_CHECK_POS;
				//State := E_MoveState.MOVE_DONE;
			ELSE
				// Điểm blend không bắt buộc robot dừng chính xác
				State := E_MoveState.MOVE_DONE;
			END_IF;

		ELSIF fbMoveP.CommandAborted THEN

			Aborted := TRUE;
			Error := TRUE;
			ErrorID_Custom := 5003;

			tMoveTimeout(IN := FALSE);

			State := E_MoveState.MOVE_ABORTED;

		ELSIF fbMoveP.Error THEN

			Error := TRUE;
			ErrorID := fbMoveP.ErrorID;
			ErrorID_Custom := 5004;

			tMoveTimeout(IN := FALSE);

			State := E_MoveState.MOVE_ERROR;

		ELSIF tMoveTimeout.Q THEN

			Timeout := TRUE;
			Error := TRUE;
			ErrorID_Custom := 5006;

			tMoveTimeout(IN := FALSE);

			State := E_MoveState.MOVE_TIMEOUT;

		END_IF;


	//========================================================
	// CHECK FINAL POSITION
	//========================================================
	E_MoveState.MOVE_CHECK_POS:

		Accepted := TRUE;

		tPosCheckDelay(
			IN := TRUE,
			PT := PosCheckDelayTime
		);

		IF tPosCheckDelay.Q THEN

			tPosCheckDelay(IN := FALSE);
// 			IF AxisGroup.m_id = SCARA_A.m_id THEN
// 				DonePosition := POU_MONITOR_ROBOT.RB1_POS;
// 			ELSE
// 				DonePosition := POU_MONITOR_ROBOT.RB2_POS;
// 			END_IF
			
			IF AxisGroup.m_id = SCARA_A.m_id THEN
				IF CoordSystem = SMC_COORD_SYSTEM.ACS THEN
					DonePosition := POU_MONITOR_ROBOT.RB1_POS_ACS;
				ELSE
					DonePosition := POU_COORDINATE_.Pos_Out_A_MCS;
				END_IF;
			ELSE
				IF CoordSystem = SMC_COORD_SYSTEM.ACS THEN
					DonePosition := POU_MONITOR_ROBOT.RB2_POS_ACS;
				ELSE
					DonePosition := POU_COORDINATE_.Pos_Out_B_MCS;
				END_IF;
				
			END_IF;

			IF F_CheckPositionReached(
				Target := PosBuf,
				//Actual := POU_MONITOR_ROBOT.RB1_POS,
				Actual := DonePosition,
				TolXYZ := GVL.MotionTolXYZ,
				TolR := GVL.MotionTolR
			) THEN
				State := E_MoveState.MOVE_DONE;

			ELSE
				Error := TRUE;
				ErrorID_Custom := 5001;
				State := E_MoveState.MOVE_ERROR;
			END_IF;
			

		END_IF;


	//========================================================
	// DONE
	//========================================================
	E_MoveState.MOVE_DONE:

		//--------------------------------------------------------
		// Giữ Done để MotionManager chắc chắn đọc được
		//--------------------------------------------------------
		Accepted := TRUE;
		Done := TRUE;
		ExecutePulse := FALSE;
		
		//--------------------------------------------------------
		// Sau khi MotionManager hạ Start và FB gốc đã rảnh,
		// wrapper được phép trở về IDLE.
		//
		// Không hạ Done tại đây; MOVE_IDLE sẽ reset ở scan sau.
		//--------------------------------------------------------
		IF NOT Start
		   AND NOT fbMoveP.Busy
		   AND NOT fbMoveP.Active
		THEN
			State := E_MoveState.MOVE_IDLE;
		END_IF;
// 		IF Release THEN
// 			Accepted := FALSE;
// 			Done := FALSE;
// 			State := E_MoveState.MOVE_IDLE;
// 			
// 		END_IF



	//========================================================
	// ERROR
	//========================================================
	E_MoveState.MOVE_ERROR:

		Error := TRUE;

		IF NOT Start THEN
			State := E_MoveState.MOVE_IDLE;
		END_IF;


	//========================================================
	// TIMEOUT
	//========================================================
	E_MoveState.MOVE_TIMEOUT:

		Error := TRUE;
		Timeout := TRUE;

		IF NOT Start THEN
			State := E_MoveState.MOVE_IDLE;
		END_IF;


	//========================================================
	// ABORTED
	//========================================================
	E_MoveState.MOVE_ABORTED:

		Error := TRUE;
		Aborted := TRUE;

		IF NOT Start THEN
			State := E_MoveState.MOVE_IDLE;
		END_IF;

END_CASE;

//============================================================
// GỌI FB GỐC MỖI SCAN
//============================================================
fbMoveP(
    AxisGroup := AxisGroup,
    Execute := ExecutePulse,

    Position := PosBuf,
    CoordSystem := CoordSystem,

    BufferMode := BufferMode,
    TransitionMode := TransMode,
    TransitionParameter := TransParam,

    VelFactor := VelFacLocal,
    AccFactor := AccFacLocal,
    JerkFactor := JerkFacLocal,
    TorqueFactor := TorqueFacLocal
);


//============================================================
// PHẢN HỒI TRẠNG THÁI FB GỐC
//============================================================
Busy := fbMoveP.Busy;
Active := fbMoveP.Active;

END_FUNCTION_BLOCK

// Just_Motion_Control_x86_64_Linux_SM_WV/Application/PRG_ROBOT/POU_MONITOR_ROBOT
PROGRAM POU_MONITOR_ROBOT
VAR
	MC_GroupReadActualPosition_1: MC_GroupReadActualPosition;
	MC_GroupReadActualPosition_2: MC_GroupReadActualPosition;
	MC_GroupReadActualVelocity_1: MC_GroupReadActualVelocity;
	MC_GroupReadActualVelocity_2: MC_GroupReadActualVelocity;
	
	MC_GroupReadActualPosition_ACS_1: MC_GroupReadActualPosition;
	MC_GroupReadActualPosition_ACS_2: MC_GroupReadActualPosition;	
	
	
	
	RB1_POS, RB2_POS, RB1_POS_ACS, RB2_POS_ACS : SM3_Robotics.SMC_POS_REF;
	
	
	
	RB1_SPEED, RB2_SPEED : SM3_Robotics.SMC_POS_REF;

	MC_ReadActualPosition_R: MC_ReadActualPosition;
	R_POS: LREAL;
	MC_ReadActualVelocity_R: MC_ReadActualVelocity;
	R_SPEED: LREAL;
	MC_GroupReadStatus_RBA: MC_GroupReadStatus;
	MC_GroupReadStatus_RBB: MC_GroupReadStatus;

	MC_GroupReadError_RBA: MC_GroupReadError;
	MC_GroupReadError_RBB: MC_GroupReadError;
	ErrorID_RBA: SM3_Robotics.SMC_ERROR;
	ErrorID_RBB: SM3_Robotics.SMC_ERROR;
	SMC_GroupReadPathDynamics_RBA: SMC_GroupReadPathDynamics;
	SMC_GroupReadPathDynamics_RBb: SMC_GroupReadPathDynamics;
	SMC_GroupReadTool_0: SMC_GroupReadTool;

	SMC_GroupReadPlanningStatistics_0: SMC_GroupReadPlanningStatistics;
END_VAR

ACT_READ();
ACT_LOGIC();
ACT_Teaching();

ACTION ACT_LOGIC:
{region "1. READ_POS_CURRENT"}
// Currern position robot
MC_GroupReadActualPosition_1.Enable := TRUE;
IF GVL.RB_A.COORD <> SMC_COORD_SYSTEM.ACS THEN
	GVL.RB_A_.CUR_X   := TO_REAL(RB1_POS.c.X);
	GVL.RB_A_.CUR_Y   := TO_REAL(RB1_POS.c.Y);
	GVL.RB_A_.CUR_Z   := TO_REAL(RB1_POS.c.Z);
	GVL.RB_A_.CUR_R   := TO_REAL(RB1_POS.c.A);
ELSIF GVL.RB_A.COORD = SMC_COORD_SYSTEM.ACS THEN
	GVL.RB_A_.CUR_X   := TO_REAL(RB1_POS.a.a0);
	GVL.RB_A_.CUR_Y   := TO_REAL(RB1_POS.a.a1);
	GVL.RB_A_.CUR_Z   := TO_REAL(RB1_POS.a.a2);
	GVL.RB_A_.CUR_R   := TO_REAL(RB1_POS.a.a3);
END_IF

/// 
MC_GroupReadActualPosition_2.Enable := TRUE;
IF GVL.RB_B.COORD <>  SMC_COORD_SYSTEM.ACS THEN
	GVL.RB_B_.CUR_X   := TO_REAL(RB2_POS.c.X);
	GVL.RB_B_.CUR_Y   := TO_REAL(RB2_POS.c.Y);
	GVL.RB_B_.CUR_Z   := TO_REAL(RB2_POS.c.Z);
	GVL.RB_B_.CUR_R   := TO_REAL(RB2_POS.c.A);
ELSIF GVL.RB_B.COORD =  SMC_COORD_SYSTEM.ACS THEN
	GVL.RB_B_.CUR_X   := TO_REAL(RB2_POS.a.a0);
	GVL.RB_B_.CUR_Y   := TO_REAL(RB2_POS.a.a1);
	GVL.RB_B_.CUR_Z   := TO_REAL(RB2_POS.a.a2);
	GVL.RB_B_.CUR_R   := TO_REAL(RB2_POS.a.a3);

END_IF
{endregion}	 
{region "2. READ_VELOCITY_CURRENT"}	 
// Currern speed robot
IF GVL.RB_A.COORD <> SMC_COORD_SYSTEM.ACS THEN
	GVL.RB_A_.CUR_SP_X   := TO_REAL(RB1_SPEED.c.X);
	GVL.RB_A_.CUR_SP_Y   := TO_REAL(RB1_SPEED.c.Y);
	GVL.RB_A_.CUR_SP_Z  := TO_REAL(RB1_SPEED.c.Z);
	GVL.RB_A_.CUR_SP_R   := TO_REAL(RB1_SPEED.c.c);
ELSIF GVL.RB_A.COORD = SMC_COORD_SYSTEM.ACS THEN
	GVL.RB_A_.CUR_SP_X   := TO_REAL(RB1_SPEED.a.a0);
	GVL.RB_A_.CUR_SP_Y   := TO_REAL(RB1_SPEED.a.a1);
	GVL.RB_A_.CUR_SP_Z  := TO_REAL(RB1_SPEED.a.a2);
	GVL.RB_A_.CUR_SP_R   := TO_REAL(RB1_SPEED.a.a3);	
END_IF
IF GVL.RB_B.COORD <> SMC_COORD_SYSTEM.ACS THEN
	GVL.RB_B_.CUR_SP_X    := TO_REAL(RB2_SPEED.c.X);
	GVL.RB_B_.CUR_SP_Y   := TO_REAL(RB2_SPEED.c.Y);
	GVL.RB_B_.CUR_SP_Z    := TO_REAL(RB2_SPEED.c.Z);
	GVL.RB_B_.CUR_SP_R   := TO_REAL(RB2_SPEED.c.c);
ELSIF GVL.RB_B.COORD = SMC_COORD_SYSTEM.ACS THEN
	GVL.RB_B_.CUR_SP_X    := TO_REAL(RB2_SPEED.a.a0);
	GVL.RB_B_.CUR_SP_Y   := TO_REAL(RB2_SPEED.a.a1);
	GVL.RB_B_.CUR_SP_Z    := TO_REAL(RB2_SPEED.a.a2);
	GVL.RB_B_.CUR_SP_R   := TO_REAL(RB2_SPEED.a.a3);	
END_IF
{endregion}
{region "3. READ_POS/VELOCITY_CURRENT_AXIS Z"}	 
// READ POSITION & SPEED axis R
// MC_ReadActualPosition_R.Enable := TRUE;
// GVL.M_R_.CUR_POS := TO_REAL(R_POS);
// GVL.M_R_.CUR_SP := TO_REAL(R_SPEED);
{endregion}
{region "4. CONDITION RUNGNING RB"}
GVL.RB_A_.Runing := POU_JOG_ROBOT.SMC_GroupJog2_1.Busy OR POU_MOTION.MOVC_A.Busy OR POU_MOTION.MOVP_A.Busy OR POU_MOTION.MOVL_A.Busy ;
GVL.RB_B_.Runing := POU_JOG_ROBOT.SMC_GroupJog2_2.Busy OR POU_MOTION.MOVC_B.Busy OR POU_MOTION.MOVP_B.Busy OR POU_MOTION.MOVL_B.Busy ;	 
{endregion}
END_ACTION

ACTION ACT_READ:
MC_GroupReadActualPosition_ACS_1(AxisGroup := SCARA_A, Enable := TRUE, CoordSystem := 0); // MC_GroupReadActualPosition
MC_GroupReadActualPosition_ACS_2(AxisGroup := SCARA_B, Enable := TRUE, CoordSystem := 0); // MC_GroupReadActualPosition
RB2_POS_ACS := MC_GroupReadActualPosition_ACS_2.Position;
MC_GroupReadActualVelocity_2(
    AxisGroup := SCARA_B,
    Enable := POU_CONTROL_ROBOT.RB_B_POWER_ON,
    CoordSystem := GVL.RB_B.COORD); // MC_GroupReadActualVelocity
RB1_POS_ACS := MC_GroupReadActualPosition_ACS_1.Position;
MC_GroupReadActualPosition_2(AxisGroup := SCARA_B, CoordSystem := GVL.RB_B.COORD); // MC_GroupReadActualPosition
RB2_POS := MC_GroupReadActualPosition_2.Position;
// READ_POSITION
MC_GroupReadActualPosition_1(AxisGroup := SCARA_A, CoordSystem := GVL.RB_A.COORD); // MC_GroupReadActualPosition
RB1_POS := MC_GroupReadActualPosition_1.Position;
// READ_VALOCITY
MC_GroupReadActualVelocity_1(
    AxisGroup := SCARA_A,
    Enable := POU_CONTROL_ROBOT.RB_A_POWER_ON,
    CoordSystem := GVL.RB_A.COORD); // MC_GroupReadActualVelocity
RB1_SPEED := MC_GroupReadActualVelocity_1.Velocity;
RB2_SPEED := MC_GroupReadActualVelocity_2.Velocity;
MC_GroupReadStatus_RBB(AxisGroup := SCARA_B, Enable := TRUE); // MC_GroupReadStatus
MC_GroupReadStatus_RBA(AxisGroup := SCARA_A, Enable := TRUE); // MC_GroupReadStatus
SMC_GroupReadTool_0(AxisGroup := SCARA_A, Execute := true, ReadMode := 2); // SMC_GroupReadTool
SMC_GroupReadPathDynamics_RBb(AxisGroup := SCARA_B, Enable := TRUE, CoordSystem := 1); // SMC_GroupReadPathDynamics
SMC_GroupReadPathDynamics_RBA(AxisGroup := SCARA_A, Enable := TRUE, CoordSystem := 1); // SMC_GroupReadPathDynamics
MC_GroupReadError_RBB(AxisGroup := SCARA_B, Enable := TRUE); // MC_GroupReadError
MC_GroupReadError_RBA(AxisGroup := SCARA_A, Enable := TRUE); // MC_GroupReadError
GVL.RB_B_.ERROR := MC_GroupReadError_RBB.Error;
GVL.RB_A_.ERROR := MC_GroupReadError_RBA.Error;
ErrorID_RBB := MC_GroupReadError_RBB.ErrorID;
ErrorID_RBA := MC_GroupReadError_RBA.ErrorID;
SMC_GroupReadPlanningStatistics_0(AxisGroup := SCARA_A, Enable := TRUE); // SMC_GroupReadPlanningStatistics
END_ACTION

ACTION ACT_Teaching:
// Teaching Robot A
IF GVL.RB_A.Manual AND 	GVL.RB_A.Comfirm_Teach AND GVL.DW_[10] > 0  THEN
	CASE GVL.RB_A.Control_w_mode OF
		0: 
			GVL_1.Point_Name_A[GVL.DW_[10]]      := GVL.HMI_A_Edit_Pos_Name;
			GVL_1.DATA_RB_A.X_POS[GVL.DW_[10]] :=  TO_REAL(LIMIT(GVL_1.DATA_RB_A.LIMIT_X_BW, GVL.RB_A_.CUR_X, GVL_1.DATA_RB_A.LIMIT_X_FW));
			GVL_1.DATA_RB_A.Y_POS[GVL.DW_[10]] :=  TO_REAL(LIMIT(GVL_1.DATA_RB_A.LIMIT_Y_BW, GVL.RB_A_.CUR_Y, GVL_1.DATA_RB_A.LIMIT_Y_FW));
			GVL_1.DATA_RB_A.Z_POS[GVL.DW_[10]] :=  TO_REAL(LIMIT(GVL_1.DATA_RB_A.LIMIT_Z_BW, GVL.RB_A_.CUR_Z, GVL_1.DATA_RB_A.LIMIT_Z_FW));
			GVL_1.DATA_RB_A.R_POS[GVL.DW_[10]] :=  TO_REAL(LIMIT(GVL_1.DATA_RB_A.LIMIT_R_BW, GVL.RB_A_.CUR_R, GVL_1.DATA_RB_A.LIMIT_R_FW));
		1:
			GVL_1.Point_Name_A[GVL.DW_[10]]      := GVL.HMI_A_Edit_Pos_Name;
			GVL_1.DATA_RB_A.X_POS[GVL.DW_[10]] := TO_REAL(GVL.RB_A_.CUR_X);
			GVL_1.DATA_RB_A.Y_POS[GVL.DW_[10]] := TO_REAL(GVL.RB_A_.CUR_Y);
			GVL_1.DATA_RB_A.Z_POS[GVL.DW_[10]] := TO_REAL(GVL.RB_A_.CUR_Z);
			GVL_1.DATA_RB_A.R_POS[GVL.DW_[10]] := TO_REAL(GVL.RB_A_.CUR_R);
	END_CASE
	GVL.RB_A.Comfirm_Teach := FALSE;
END_IF


IF GVL.RB_B.Manual AND GVL.RB_B.Comfirm_Teach AND GVL.DW_[12] > 0 THEN
    CASE GVL.RB_B.Control_w_mode OF
        0:
            GVL_1.Point_Name_B[GVL.DW_[12]] := GVL.HMI_B_Edit_Pos_Name;
            GVL_1.DATA_RB_B.X_POS[GVL.DW_[12]] := TO_REAL(LIMIT(GVL_1.DATA_RB_B.LIMIT_X_BW, GVL.RB_B_.CUR_X, GVL_1.DATA_RB_B.LIMIT_X_FW));
            GVL_1.DATA_RB_B.Y_POS[GVL.DW_[12]] := TO_REAL(LIMIT(GVL_1.DATA_RB_B.LIMIT_Y_BW, GVL.RB_B_.CUR_Y, GVL_1.DATA_RB_B.LIMIT_Y_FW));
            GVL_1.DATA_RB_B.Z_POS[GVL.DW_[12]] := TO_REAL(LIMIT(GVL_1.DATA_RB_B.LIMIT_Z_BW, GVL.RB_B_.CUR_Z, GVL_1.DATA_RB_B.LIMIT_Z_FW));
            GVL_1.DATA_RB_B.R_POS[GVL.DW_[12]] := TO_REAL(LIMIT(GVL_1.DATA_RB_B.LIMIT_R_BW, GVL.RB_B_.CUR_R, GVL_1.DATA_RB_B.LIMIT_R_FW));
        1:
            GVL_1.Point_Name_B[GVL.DW_[12]] := GVL.HMI_B_Edit_Pos_Name;
            GVL_1.DATA_RB_B.X_POS[GVL.DW_[12]] := TO_REAL(GVL.RB_B_.CUR_X);
            GVL_1.DATA_RB_B.Y_POS[GVL.DW_[12]] := TO_REAL(GVL.RB_B_.CUR_Y);
            GVL_1.DATA_RB_B.Z_POS[GVL.DW_[12]] := TO_REAL(GVL.RB_B_.CUR_Z);
            GVL_1.DATA_RB_B.R_POS[GVL.DW_[12]] := TO_REAL(GVL.RB_B_.CUR_R);
    END_CASE;
    GVL.RB_B.Comfirm_Teach := FALSE;
END_IF;

	
// // Teaching Robot B
// IF GVL.RB_B.Manual AND 	GVL.RB_B.Comfirm_Teach AND GVL.DW_[12] > 0  THEN
// 	CASE GVL.RB_B.Control_w_mode OF
// 		0:	
// 			//GVL_1.Point_Name_B[GVL.DW_[12]]      := GVL.HMI_B_Edit_Pos_Name;
// 			GVL_1.DATA_RB_B.X_POS[GVL.DW_[12]] :=  TO_REAL(LIMIT(GVL_1.DATA_RB_B.LIMIT_X_BW, GVL.RB_B_.CUR_X, GVL_1.DATA_RB_B.LIMIT_X_FW));
// 			GVL_1.DATA_RB_B.Y_POS[GVL.DW_[12]] :=  TO_REAL(LIMIT(GVL_1.DATA_RB_B.LIMIT_Y_BW, GVL.RB_B_.CUR_Y, GVL_1.DATA_RB_B.LIMIT_Y_FW));
// 			GVL_1.DATA_RB_B.Z_POS[GVL.DW_[12]] :=  TO_REAL(LIMIT(GVL_1.DATA_RB_B.LIMIT_Z_BW, GVL.RB_B_.CUR_Z, GVL_1.DATA_RB_B.LIMIT_Z_FW));
// 			GVL_1.DATA_RB_B.R_POS[GVL.DW_[12]] :=  TO_REAL(LIMIT(GVL_1.DATA_RB_B.LIMIT_R_BW, GVL.RB_B_.CUR_R, GVL_1.DATA_RB_B.LIMIT_R_FW));	
// 		1:
// 			GVL_1.DATA_RB_B.X_POS[GVL.DW_[12]] := TO_REAL(GVL.RB_B_.CUR_X);
// 			GVL_1.DATA_RB_B.Y_POS[GVL.DW_[12]] := TO_REAL(GVL.RB_B_.CUR_Y);
// 			GVL_1.DATA_RB_b.Z_POS[GVL.DW_[12]] := TO_REAL(GVL.RB_B_.CUR_Z);
// 			GVL_1.DATA_RB_B.R_POS[GVL.DW_[12]] := TO_REAL(GVL.RB_B_.CUR_R);
// 	END_CASE	
// GVL.RB_B.Comfirm_Teach := FALSE;
// END_IF
END_ACTION

END_PROGRAM

// Just_Motion_Control_x86_64_Linux_SM_WV/Application/PRG_ROBOT/POU_JOG_ROBOT
PROGRAM POU_JOG_ROBOT
VAR // funtion 
	SMC_GroupJog2_1: SMC_GroupJog2;
	SMC_GroupJog2_2: SMC_GroupJog2;
	MC_JOG_R: MC_Jog;
	CoordSystem_A: SM3_Robotics.SMC_COORD_SYSTEM;
	CoordSystem_B: SM3_Robotics.SMC_COORD_SYSTEM;
END_VAR
VAR
	Jog_FW_A: ARRAY [0..(SMC_RCNST.MAX_AXES - 1)] OF BOOL;
	Jog_BW_A: ARRAY [0..(SMC_RCNST.MAX_AXES - 1)] OF BOOL;
	Jog_FW_B: ARRAY [0..(SMC_RCNST.MAX_AXES - 1)] OF BOOL;
	Jog_BW_B: ARRAY [0..(SMC_RCNST.MAX_AXES - 1)] OF BOOL;
	
	FOCUS_JOG_A, FOCUS_JOG_B : BOOL;	
	Jog_FW, Jog_BW : BOOL;
	
	
END_VAR
VAR // added by the converter: edge detectors and wires of the graphical bodies
    _w1, _w2, _w3, _w4, _w5, _w6, _w7, _w8 : LREAL;
END_VAR

ACT_JOG();
ACT_LOGIC_A();
ACT_LOGIC_B();
// ACT_LOGIC_R();

ACTION ACT_JOG:
_w1 := TO_LREAL(GVL.RB_A.DEC);
_w2 := TO_LREAL(GVL.RB_A.ACC);
_w3 := TO_LREAL(GVL.RB_A.SPEED);
_w4 := TO_LREAL(GVL.RB_A.JERK);
_w5 := TO_LREAL(GVL.Fac_Vel_Set_A);
_w6 := TO_LREAL(GVL.Fac_Torque_Set_A);
_w7 := TO_LREAL(GVL.Fac_Acc_Set_A);
_w8 := TO_LREAL(GVL.Fac_Jerk_Set_A);
SMC_GroupJog2_2(
    AxisGroup := SCARA_B,
    Forward := Jog_FW_B,
    Backward := Jog_BW_B,
    MaxLinearDistance := GVL_1.DATA_RB_B.LinearDistanceJog,
    MaxAngularDistance := GVL_1.DATA_RB_B.AngularDistanceJog,
    Velocity := TO_LREAL(GVL.RB_B.SPEED),
    Acceleration := TO_LREAL(GVL.RB_B.ACC),
    Deceleration := TO_LREAL(GVL.RB_B.DEC),
    Jerk := TO_LREAL(GVL.RB_b.JERK),
    VelFactor := TO_LREAL(GVL.Fac_Vel_Set_B),
    AccFactor := TO_LREAL(GVL.Fac_Acc_Set_B),
    JerkFactor := TO_LREAL(GVL.Fac_Jerk_Set_B),
    TorqueFactor := TO_LREAL(GVL.Fac_Torque_Set_B),
    CoordSystem := CoordSystem_B); // SMC_GroupJog2
// JOG_ROBOT
SMC_GroupJog2_1(
    AxisGroup := SCARA_A,
    Forward := Jog_FW_A,
    Backward := Jog_BW_A,
    MaxLinearDistance := GVL_1.DATA_RB_A.LinearDistanceJog,
    MaxAngularDistance := GVL_1.DATA_RB_A.AngularDistanceJog,
    Velocity := _w3,
    Acceleration := _w2,
    Deceleration := _w1,
    Jerk := _w4,
    VelFactor := _w5,
    AccFactor := _w7,
    JerkFactor := _w8,
    TorqueFactor := _w6,
    CoordSystem := CoordSystem_A); // SMC_GroupJog2
END_ACTION

ACTION ACT_LOGIC_A:
{region "1. Logic Jog"}
// JOG ROBOT A
IF GVL.RB_A.Jog_continue THEN
Jog_FW_A[0]:= GVL.RB_A.JOG_X_FW ;
Jog_FW_A[1]:= GVL.RB_A.JOG_Y_FW ;
Jog_FW_A[2]:= GVL.RB_A.JOG_Z_FW ;

Jog_BW_A[0]:= GVL.RB_A.JOG_X_BW ;
Jog_BW_A[1]:= GVL.RB_A.JOG_Y_BW ;
Jog_BW_A[2]:= GVL.RB_A.JOG_Z_BW ;

	IF  gvl.RB_A.ABC_as_ACS OR GVL.RB_A.COORD = 0 THEN
		Jog_FW_A[3]:= GVL.RB_A.JOG_R_FW ;	 
		Jog_BW_A[3]:= GVL.RB_A.JOG_R_BW ;	
	ELSIF NOT gvl.RB_A.ABC_as_ACS AND GVL.RB_A.COORD <> 0 THEN
		Jog_FW_A[5]:= GVL.RB_A.JOG_R_FW ;	 
		Jog_BW_A[5]:= GVL.RB_A.JOG_R_BW ;  
	END_IF;			   
END_IF;

FOCUS_JOG_A := Jog_FW_A[0] OR Jog_FW_A[1] OR Jog_FW_A[2] OR Jog_FW_A[3] OR Jog_FW_A[4] OR Jog_FW_A[5]
			OR Jog_BW_A[0] OR Jog_BW_A[1] OR Jog_BW_A[2] OR Jog_BW_A[3] OR Jog_BW_A[4] OR Jog_BW_A[5] ;

// CONDITION
IF GVL.RB_A.Manual AND GVL.RB_A_.Ready AND ( GVL.RB_A_.SAFETY_CHECK OR gvl.RB_A.Control_w_mode = 1) AND FOCUS_JOG_A THEN
	SMC_GroupJog2_1.Enable := TRUE;
	ELSE
	SMC_GroupJog2_1.Enable := FALSE;	
END_IF

SMC_GroupJog2_1.ABC_as_ACS := gvl.RB_A.ABC_as_ACS; // true giữ nguyên tool, false : tool quay theo
{endregion}
{region "2. Control Parameter"}
/// CONTROL SPEED
IF GVL.RB_A.Auto THEN
	GVL.RB_A.ACC := GVL_1.DATA_RB_A.MOTION_ACC;
	GVL.RB_A.DEC := GVL_1.DATA_RB_A.MOTION_DEC;
	GVL.RB_A.JERK := GVL_1.DATA_RB_A.MOTION_JERK;
ELSE
	GVL.RB_A.ACC :=  GVL_1.DATA_RB_A.MOTION_ACC_MAN;
	GVL.RB_A.DEC := GVL_1.DATA_RB_A.MOTION_DEC_MAN;
	GVL.RB_A.JERK := GVL_1.DATA_RB_A.MOTION_JERK_MAN;
END_IF;
IF GVL.RB_A.Control_w_speed = 2 THEN
	IF GVL.RB_A.Auto THEN
		GVL.RB_A.SPEED := GVL_1.DATA_RB_A.SPEED_HIGH;
	ELSE
		GVL.RB_A.SPEED := GVL.RB_A_Man.SPEED_High_Man;
	END_IF;
ELSIF GVL.RB_A.Control_w_speed = 1 THEN
	IF GVL.RB_A.Auto THEN
		GVL.RB_A.SPEED := GVL_1.DATA_RB_A.SPEED_MID;
	ELSE
		GVL.RB_A.SPEED := GVL_1.DATA_RB_A.SPEED_MID_MAN;
	END_IF;
ELSE
	IF GVL.RB_A.Auto THEN
		GVL.RB_A.SPEED := GVL_1.DATA_RB_A.SPEED_LOW;	
	ELSE
		GVL.RB_A.SPEED := GVL_1.DATA_RB_A.SPEED_LOW_MAN;
	END_IF;
END_IF
{endregion}	 
	 
{region "3. Coordinate System"}
CASE GVL.RB_A.COORD OF
	0:
		CoordSystem_A := SM3_Robotics.SMC_COORD_SYSTEM.ACS;
	1:
		CoordSystem_A := SM3_Robotics.SMC_COORD_SYSTEM.MCS;	 
	2:
		CoordSystem_A := SM3_Robotics.SMC_COORD_SYSTEM.WCS;	
	3:
		CoordSystem_A := SM3_Robotics.SMC_COORD_SYSTEM.PCS_1;			 
	4:
		CoordSystem_A := SM3_Robotics.SMC_COORD_SYSTEM.PCS_2;
	5:
		CoordSystem_A := SM3_Robotics.SMC_COORD_SYSTEM.MCS; 
		//CoordSystem_A := SM3_Robotics.SMC_COORD_SYSTEM.TCS;				  
END_CASE

{endregion}
END_ACTION

ACTION ACT_LOGIC_B:
{region "1. Logic Jog"}
// JOG ROBOT B
IF GVL.RB_B.Jog_continue THEN
Jog_FW_B[0]:= GVL.RB_B.JOG_X_FW ;
Jog_FW_B[1]:= GVL.RB_B.JOG_Y_FW ;
Jog_FW_B[2]:= GVL.RB_B.JOG_Z_FW ;


Jog_BW_B[0]:= GVL.RB_B.JOG_X_BW ;
Jog_BW_B[1]:= GVL.RB_B.JOG_Y_BW ;
Jog_BW_B[2]:= GVL.RB_B.JOG_Z_BW ;

	 
	IF  gvl.RB_B.ABC_as_ACS OR GVL.RB_B.COORD = 0 THEN
		Jog_FW_B[3]:= GVL.RB_B.JOG_R_FW ;	 
		Jog_BW_B[3]:= GVL.RB_B.JOG_R_BW ;	
	ELSIF NOT gvl.RB_b.ABC_as_ACS AND GVL.RB_b.COORD <> 0 THEN
		Jog_FW_b[5]:= GVL.RB_b.JOG_R_FW ;	 
		Jog_BW_b[5]:= GVL.RB_b.JOG_R_BW ;  
	END_IF;		 			   
END_IF;

FOCUS_JOG_B := Jog_FW_B[0] OR Jog_FW_B[1] OR Jog_FW_B[2] OR Jog_FW_B[3] OR Jog_FW_B[4] OR Jog_FW_B[5]
			OR Jog_BW_B[0] OR Jog_BW_B[1] OR Jog_BW_B[2] OR Jog_BW_B[3] OR Jog_BW_B[4] OR Jog_BW_B[5];

// CONDITION
IF GVL.RB_b.Manual AND GVL.RB_b_.Ready AND (GVL.RB_b_.SAFETY_CHECK OR gvl.RB_B.Control_w_mode = 1) AND FOCUS_JOG_B THEN
	SMC_GroupJog2_2.Enable := TRUE; 
	ELSE
	SMC_GroupJog2_2.Enable := FALSE;	
END_IF

SMC_GroupJog2_2.ABC_as_ACS := gvl.RB_B.ABC_as_ACS; // true giữ nguyên tool, false : tool quay theo
{endregion}
{region "2. Control Parameter"}	 
/// CONTROL SPEED
IF GVL.RB_B.Auto THEN
	GVL.RB_B.ACC := GVL_1.DATA_RB_B.MOTION_ACC;
	GVL.RB_B.DEC := GVL_1.DATA_RB_B.MOTION_DEC;
	GVL.RB_B.JERK := GVL_1.DATA_RB_B.MOTION_JERK;
ELSE
	GVL.RB_B.ACC := GVL_1.DATA_RB_B.MOTION_ACC_MAN;
	GVL.RB_B.DEC := GVL_1.DATA_RB_B.MOTION_DEC_MAN;
	GVL.RB_B.JERK := GVL_1.DATA_RB_B.MOTION_JERK_MAN; 
END_IF	 
IF GVL.RB_b.Control_w_speed = 2 THEN
	IF GVL.RB_B.Auto THEN
		GVL.RB_B.SPEED := GVL_1.DATA_RB_B.SPEED_HIGH;
	ELSE
		GVL.RB_B.SPEED := GVL_1.DATA_RB_B.SPEED_HIGH_MAN;	 
	END_IF
ELSIF GVL.RB_b.Control_w_speed = 1 THEN
	IF GVL.RB_B.Auto THEN
		GVL.RB_B.SPEED := GVL_1.DATA_RB_B.SPEED_MID;
	ELSE
		GVL.RB_B.SPEED := GVL_1.DATA_RB_B.SPEED_MID_MAN;	 
	END_IF
ELSE
	IF GVL.RB_B.Auto THEN
		GVL.RB_B.SPEED := GVL_1.DATA_RB_B.SPEED_LOW;	
	ELSE
		GVL.RB_B.SPEED := GVL_1.DATA_RB_B.SPEED_LOW_MAN;	 
	END_IF
END_IF
{endregion}
{region "3. Coordinate System"}
CASE GVL.RB_B.COORD OF
	0:
		CoordSystem_B := SM3_Robotics.SMC_COORD_SYSTEM.ACS;
	1:
		CoordSystem_B := SM3_Robotics.SMC_COORD_SYSTEM.MCS;	 
	2:
		CoordSystem_B := SM3_Robotics.SMC_COORD_SYSTEM.WCS;	
	3:
		CoordSystem_B := SM3_Robotics.SMC_COORD_SYSTEM.PCS_1;			 
	4:
		CoordSystem_B := SM3_Robotics.SMC_COORD_SYSTEM.PCS_2;
	5:
		CoordSystem_B := SM3_Robotics.SMC_COORD_SYSTEM.MCS;	
		//CoordSystem_B := SM3_Robotics.SMC_COORD_SYSTEM.TCS;				  
END_CASE

{endregion}
END_ACTION

ACTION ACT_LOGIC_R:
// IF GVL.M_R.JOG_FW AND GVL.M_R_.SAFETY_CHECK AND GVL.M_R.Manual THEN
// 	Jog_FW := TRUE;
// 	ELSE
// 	Jog_FW := FALSE;	
// END_IF
// 
// IF GVL.M_R.JOG_BW AND (GVL.M_R_.SAFETY_CHECK OR gvl.M_R.Control_w_mode = 1) AND GVL.M_R.Manual THEN
// 	Jog_BW := TRUE;
// 	ELSE
// 	Jog_BW := FALSE;	
// END_IF

/// CONTROL SPEED
// GVL.M_R.ACC := GVL_1.DATA_M_R.MOTION_ACC;
// GVL.M_R.DEC := GVL_1.DATA_M_R.MOTION_DEC;
// GVL.M_R.JERK := GVL_1.DATA_M_R.MOTION_JERK;
// IF GVL.M_R.Control_w_speed = 2 THEN
// 	GVL.M_R.SPEED := GVL_1.DATA_M_R.SPEED_HIGH;
// ELSIF GVL.M_R.Control_w_speed = 1 THEN
// 	GVL.M_R.SPEED := GVL_1.DATA_M_R.SPEED_MID;
// ELSE
// 	GVL.M_R.SPEED := GVL_1.DATA_M_R.SPEED_LOW;	
// END_IF
END_ACTION

END_PROGRAM

// Just_Motion_Control_x86_64_Linux_SM_WV/Application/PRG_ROBOT/POU_CONTROL_ROBOT
PROGRAM POU_CONTROL_ROBOT
VAR
	
	// DEFIND FUNTION ROBOT
	SMC_GroupPower_1: SMC_GroupPower;
	SMC_GroupPower_2: SMC_GroupPower;
	SMC3_BrakeControl_A0: SMC3_BrakeControl;
	SMC3_BrakeControl_A1: SMC3_BrakeControl;
	SMC3_BrakeControl_A2: SMC3_BrakeControl;
	SMC3_BrakeControl_A3: SMC3_BrakeControl;
	SMC3_BrakeControl_B0: SMC3_BrakeControl;
	SMC3_BrakeControl_B1: SMC3_BrakeControl;
	SMC3_BrakeControl_B2: SMC3_BrakeControl;
	SMC3_BrakeControl_B3: SMC3_BrakeControl;
	MC_GroupEnable_1: MC_GroupEnable;
	MC_GroupEnable_2: MC_GroupEnable;
	MC_GroupReset_1: MC_GroupReset;
	MC_GroupReset_2: MC_GroupReset;
	MC_Power_R: MC_Power;
	MC_Home_R_MAIN : MC_Home;
	MC_Reset_R: MC_Reset;
	MC_Reset_M1: MC_Reset;
	MC_Reset_M2: MC_Reset;
	MC_Reset_M3: MC_Reset;
	MC_Reset_M4: MC_Reset;
	
	
	//IdError: SM3_Robotics.SMC_ERROR;
	MC_Reset_M21: MC_Reset;
	MC_Reset_M22: MC_Reset;
	MC_Reset_M23: MC_Reset;
	MC_Reset_M24: MC_Reset;
	//RBA_compatibiloty: SM3_Robotics.SMC_AXIS_GROUP_COMPATIBILITY_OPTIONS;
	//RBb_compatibiloty: SM3_Robotics.SMC_AXIS_GROUP_COMPATIBILITY_OPTIONS;
	MC_GroupDisable_1: MC_GroupDisable;
	MC_GroupDisable_2: MC_GroupDisable;
	
	
	SMC_GroupSetAxisLimitFactors_A: SMC_GroupSetAxisLimitFactors;
	VEL_A , ACC_A, DEC_A, JERK_A, TORQUE_A : ARRAY [0..(SMC_RCNST.MAX_AXES - 1)] OF LREAL;
	SMC_GroupSetAxisLimitFactors_B: SMC_GroupSetAxisLimitFactors;
	VEL_B , ACC_B, DEC_B, JERK_B, TORQUE_B : ARRAY [0..(SMC_RCNST.MAX_AXES - 1)] OF LREAL;

	MC_Power_AX6: MC_Power;
	MC_ReadActualPosition_AX6: MC_ReadActualPosition;
	MC_TrackConveyorBelt_0: MC_TrackConveyorBelt;
	MC_ReadActualVelocity_AX6: MC_ReadActualVelocity;
	MC_ReadActualPosition_0: MC_ReadActualPosition;
	SMC_GroupSetPathTolerance_0: SMC_GroupSetPathTolerance;
	MC_Power_0: MC_Power;
	MC_MoveVelocity_0: MC_MoveVelocity;
	MC_Reset_AX6: MC_Reset;
END_VAR
VAR
	
	RB_A_POWER_ON, RB_B_POWER_ON : BOOL;
	R_POWER_ON: BOOL;
	CASE_A_ON, CASE_A_OFF, CASE_B_ON, CASE_B_OFF, CASE_R_ON, CASE_R_OFF : INT;

	
	I : INT;
	bResetEtherCAT: BOOL;
	
	stMaxAxisLag : TRAFO.AXISPOS_REF;
	J1_PosError,J2_PosError,J1_VelError,J2_VelError: LREAL;
END_VAR

ACT_LOGIC();
ACT_POWER();
ACT_Reset();
ACT_SET_DYNAMICLIMITS();

ACTION ACT_LOGIC:
// ROBOT 1
IF GVL.RB_A.Power AND NOT SMC_GroupPower_1.Status AND NOT SMC_GroupPower_1.Busy THEN // POWER ROBOT 1
	CASE CASE_A_ON OF
	0:
		SMC_GroupPower_1.Enable := 0;
		SMC_GroupPower_1.bDriveStart := 0;
		SMC_GroupPower_1.bRegulatorOn := 0;
		CASE_A_ON := 5;
		
	5:
		SMC_GroupPower_1.Enable := 1;
		SMC_GroupPower_1.bDriveStart := 1;
		SMC_GroupPower_1.bRegulatorOn := 1;

	
	END_CASE
ELSIF NOT GVL.RB_A.Power AND SMC_GroupPower_1.Status AND NOT SMC_GroupPower_1.Busy THEN
		CASE CASE_A_OFF OF
	0:
		SMC_GroupPower_1.Enable := 0;
		SMC_GroupPower_1.bDriveStart := 0;
		SMC_GroupPower_1.bRegulatorOn := 0;
		CASE_A_OFF := 5;
		
	5:
		SMC_GroupPower_1.Enable := 1;
		SMC_GroupPower_1.bDriveStart := 0;
		SMC_GroupPower_1.bRegulatorOn := 1;
	END_CASE
ELSE
	CASE_A_ON := 0;
	CASE_A_OFF := 0;
	SMC_GroupPower_1.Enable := 0;
	SMC_GroupPower_1.bDriveStart := 0;
	SMC_GroupPower_1.bRegulatorOn := 0;;
END_IF



IF GVL.RB_A.Enable AND RB_A_POWER_ON THEN // ENABLE ROBOT 1
	MC_GroupEnable_1.Execute := 1;
	MC_GroupDisable_1.Execute := 0;
	ELSE
	MC_GroupEnable_1.Execute := 0;
	MC_GroupDisable_1.Execute := 1;
END_IF

IF NOT GVL.RB_Signal_In.HMI_EMG THEN
	MC_GroupEnable_1.Execute := 0;
	MC_GroupDisable_1.Execute := 1;
	GVL.RB_A.Power := 0;
	GVL.RB_A.Enable := 0;
END_IF
IF GVL.RB_A.BK1 THEN // A0 BRAKE
	SMC3_BrakeControl_A0.bExecute := 1;
	SMC3_BrakeControl_A0.eSetBrake := 1;
	ELSE
	SMC3_BrakeControl_A0.bExecute := 0;
	SMC3_BrakeControl_A0.eSetBrake := 0;
END_IF
IF GVL.RB_A.BK2 THEN // A1 BRAKE
	SMC3_BrakeControl_A1.bExecute := 1;
	SMC3_BrakeControl_A1.eSetBrake := 1;
	ELSE
	SMC3_BrakeControl_A1.bExecute := 0;
	SMC3_BrakeControl_A1.eSetBrake := 0;
END_IF
IF GVL.RB_A.BK3 THEN // A2 BRAKE
	SMC3_BrakeControl_A2.bExecute := 1;
	SMC3_BrakeControl_A2.eSetBrake := 1;
	ELSE
	SMC3_BrakeControl_A2.bExecute := 0;
	SMC3_BrakeControl_A2.eSetBrake := 0;
END_IF
IF GVL.RB_A.BK4 THEN // A3 BRAKE
	SMC3_BrakeControl_A3.bExecute := 1;
	SMC3_BrakeControl_A3.eSetBrake := 1;
	ELSE
	SMC3_BrakeControl_A3.bExecute := 0;
	SMC3_BrakeControl_A3.eSetBrake := 0;
END_IF

///////////////////////////////////////////////////////////////////////////////////////////////////////////

// ROBOT 2
IF GVL.RB_B.Power AND NOT SMC_GroupPower_2.Status AND NOT SMC_GroupPower_2.Busy THEN // POWER ROBOT 2
	CASE CASE_B_ON OF
	0:
		SMC_GroupPower_2.Enable := 0;
		SMC_GroupPower_2.bDriveStart := 0;
		SMC_GroupPower_2.bRegulatorOn := 0;
		CASE_B_ON := 5;
		
	5:
		SMC_GroupPower_2.Enable := 1;
		SMC_GroupPower_2.bDriveStart := 1;
		SMC_GroupPower_2.bRegulatorOn := 1;
	END_CASE
ELSIF NOT GVL.RB_B.Power AND SMC_GroupPower_2.Status AND NOT SMC_GroupPower_2.Busy THEN
		CASE CASE_B_OFF OF
	0:
		SMC_GroupPower_2.Enable := 0;
		SMC_GroupPower_2.bDriveStart := 0;
		SMC_GroupPower_2.bRegulatorOn := 0;
		CASE_b_OFF := 5;
		
	5:
		SMC_GroupPower_2.Enable := 1;
		SMC_GroupPower_2.bDriveStart := 0;
		SMC_GroupPower_2.bRegulatorOn := 1;
	END_CASE
ELSE
	CASE_b_ON := 0;
	CASE_b_OFF := 0;
	SMC_GroupPower_2.Enable := 0;
	SMC_GroupPower_2.bDriveStart := 0;
	SMC_GroupPower_2.bRegulatorOn := 0;;
END_IF
IF RB_B_POWER_ON AND GVL.RB_B.Enable THEN // ENABLE ROBOT 2
	MC_GroupEnable_2.Execute := 1;
	MC_GroupDisable_2.Execute := 0;
	ELSE
	MC_GroupEnable_2.Execute := 0;
	MC_GroupDisable_2.Execute := 1;
END_IF

IF NOT GVL.RB_Signal_In.HMI_EMG THEN
	MC_GroupEnable_2.Execute := 0;
	MC_GroupDisable_2.Execute := 1;
	GVL.RB_B.Power := 0;
	GVL.RB_B.Enable := 0;
END_IF

IF GVL.RB_B.BK1 THEN // B0 BRAKE
	SMC3_BrakeControl_B0.bExecute := 1;
	SMC3_BrakeControl_B0.eSetBrake := 1;
	ELSE
	SMC3_BrakeControl_B0.bExecute := 0;
	SMC3_BrakeControl_B0.eSetBrake := 0;
END_IF
IF GVL.RB_B.BK2 THEN // B1 BRAKE
	SMC3_BrakeControl_B1.bExecute := 1;
	SMC3_BrakeControl_B1.eSetBrake := 1;
	ELSE
	SMC3_BrakeControl_B1.bExecute := 0;
	SMC3_BrakeControl_B1.eSetBrake := 0;
END_IF
IF GVL.RB_B.BK3 THEN // B2 BRAKE
	SMC3_BrakeControl_B2.bExecute := 1;
	SMC3_BrakeControl_B2.eSetBrake := 1;
	ELSE
	SMC3_BrakeControl_B2.bExecute := 0;
	SMC3_BrakeControl_B2.eSetBrake := 0;
END_IF
IF GVL.RB_B.BK4 THEN // B3 BRAKE
	SMC3_BrakeControl_B3.bExecute := 1;
	SMC3_BrakeControl_B3.eSetBrake := 1;
	ELSE
	SMC3_BrakeControl_B3.bExecute := 0;
	SMC3_BrakeControl_B3.eSetBrake := 0;
END_IF

///////////////////////////////////////////////////////////////////////////////////////////////////////////

// R_MAIN
// IF GVL.M_R.Power THEN // POWER R MAIN
// 	MC_Power_R.Enable := 1;
// 	MC_Power_R.bDriveStart := 1;
// 	MC_Power_R.bRegulatorOn := 1;
// 	ELSE
// 	MC_Power_R.Enable := 0;
// 	MC_Power_R.bDriveStart := 0;
// 	MC_Power_R.bRegulatorOn := 0;	
// END_IF
// IF GVL.M_R.Power AND NOT MC_Power_R.Status AND NOT MC_Power_R.Busy THEN // POWER ROBOT 1
// 	CASE CASE_R_ON OF
// 	0:
// 		MC_Power_R.Enable := 0;
// 		MC_Power_R.bDriveStart := 0;
// 		MC_Power_R.bRegulatorOn := 0;
// 		CASE_R_ON := 5;
// 		
// 	5:
// 		MC_Power_R.Enable := 1;
// 		MC_Power_R.bDriveStart := 1;
// 		MC_Power_R.bRegulatorOn := 1;
// 
// 	
// 	END_CASE
// ELSIF NOT GVL.M_R.Power AND MC_Power_R.Status AND NOT MC_Power_R.Busy THEN
// 		CASE CASE_R_OFF OF
// 	0:
// 		MC_Power_R.Enable := 0;
// 		MC_Power_R.bDriveStart := 0;
// 		MC_Power_R.bRegulatorOn := 0;
// 		CASE_R_OFF := 5;
// 		
// 	5:
// 		MC_Power_R.Enable := 1;
// 		MC_Power_R.bDriveStart := 0;
// 		MC_Power_R.bRegulatorOn := 1;
// 	END_CASE
// ELSE
// 	CASE_R_ON := 0;
// 	CASE_R_OFF := 0;
// 	MC_Power_R.Enable := 0;
// 	MC_Power_R.bDriveStart := 0;
// 	MC_Power_R.bRegulatorOn := 0;;
// END_IF
END_ACTION

ACTION ACT_POWER:
SMC3_BrakeControl_A3(Axis := A3); // SMC3_BrakeControl
MC_Reset_M2(Axis := A1); // MC_Reset
SMC3_BrakeControl_B0(Axis := B0); // SMC3_BrakeControl
SMC3_BrakeControl_A1(Axis := A1); // SMC3_BrakeControl
// POWER ROBOT:
SMC_GroupPower_1(AxisGroup := SCARA_A); // SMC_GroupPower
RB_A_POWER_ON := SMC_GroupPower_1.Status;
SMC_GroupPower_2(AxisGroup := SCARA_B); // SMC_GroupPower
RB_B_POWER_ON := SMC_GroupPower_2.Status;
SMC3_BrakeControl_B1(Axis := B1); // SMC3_BrakeControl
MC_Reset_M21(Axis := B0); // MC_Reset
MC_Reset_M22(Axis := B1); // MC_Reset
MC_Reset_M3(Axis := A2); // MC_Reset
MC_GroupEnable_2(AxisGroup := SCARA_B); // MC_GroupEnable
GVL.RB_B_.Ready := MC_GroupEnable_2.Done;
MC_Reset_M23(Axis := B2); // MC_Reset
MC_Reset_AX6(Axis := AXIS_6); // MC_Reset
SMC_GroupSetPathTolerance_0(
    AxisGroup := SCARA_A,
    MaxPositionLag := 3,
    MaxOrientationLag := 5.0,
    MaxAxisLag := stMaxAxisLag); // SMC_GroupSetPathTolerance
MC_Reset_M4(Axis := A3); // MC_Reset
MC_GroupDisable_1(AxisGroup := SCARA_A); // MC_GroupDisable
MC_GroupDisable_2(AxisGroup := SCARA_B); // MC_GroupDisable
SMC3_BrakeControl_B2(Axis := B2); // SMC3_BrakeControl
SMC3_BrakeControl_B3(Axis := B3); // SMC3_BrakeControl
// CONTROL BRAKE MOTOR:
SMC3_BrakeControl_A0(Axis := A0); // SMC3_BrakeControl
MC_GroupReset_2(AxisGroup := SCARA_B); // MC_GroupReset
SMC3_BrakeControl_A2(Axis := A2); // SMC3_BrakeControl
// ENABLE_ROBOT
MC_GroupEnable_1(AxisGroup := SCARA_A); // MC_GroupEnable
GVL.RB_A_.Ready := MC_GroupEnable_1.Done;
// RESET_ROBOT
MC_GroupReset_1(AxisGroup := SCARA_A); // MC_GroupReset
MC_Reset_M1(Axis := A0); // MC_Reset
MC_Reset_M24(Axis := B3); // MC_Reset
MC_Power_0(Axis := B1); // MC_Power
MC_MoveVelocity_0(Axis := A0, Execute := GVL.RB_A.JOG_X_FW); // MC_MoveVelocity
END_ACTION

ACTION ACT_Reset:
IF GVL.RB_A.Reset OR GVL.X[8] THEN
	MC_GroupReset_1.Execute := TRUE;
	MC_Reset_M1.Execute := TRUE;
	MC_Reset_M2.Execute := TRUE;
	MC_Reset_M3.Execute := TRUE;
	MC_Reset_M4.Execute := TRUE;
	MC_Reset_AX6.Execute := TRUE;
ELSE
	MC_GroupReset_1.Execute := FALSE;
	MC_Reset_M1.Execute := FALSE;
	MC_Reset_M2.Execute := FALSE;
	MC_Reset_M3.Execute := FALSE;
	MC_Reset_M4.Execute := FALSE;	
	MC_Reset_AX6.Execute := FALSE;
END_IF

/// robto 2

IF GVL.RB_B.Reset OR GVL.X[8] THEN
	MC_GroupReset_2.Execute := TRUE;
	MC_Reset_M21.Execute := TRUE;
	MC_Reset_M22.Execute := TRUE;
	MC_Reset_M23.Execute := TRUE;
	MC_Reset_M24.Execute := TRUE;
ELSE
	MC_GroupReset_2.Execute := FALSE;
	MC_Reset_M21.Execute := FALSE;
	MC_Reset_M22.Execute := FALSE;
	MC_Reset_M23.Execute := FALSE;
	MC_Reset_M24.Execute := FALSE;	
END_IF

// Khi nhấn nút Reset lỗi EtherCAT trên HMI/PLC
IF bResetEtherCAT THEN
    EtherCAT_Master_SoftMotion.xRestart := TRUE;
    bResetEtherCAT := FALSE;
END_IF
END_ACTION

ACTION ACT_SET_DYNAMICLIMITS:
WHILE GVL.HMI_MAIN.Enable_Dynamics_Limit DO	
FOR I := 0 TO 3 BY 1 DO
	VEL_A[I]	:= GVL_1.DATA_RB_A.MAX_VEL;
	ACC_A[I]	:= GVL_1.DATA_RB_A.MAX_ACC;
	JERK_A[I]	:= GVL_1.DATA_RB_A.MAX_JERK;
	TORQUE_A[I]	:= GVL_1.DATA_RB_A.MAX_TOQUE;
	
	VEL_B[I]	:= GVL_1.DATA_RB_B.MAX_VEL;
	ACC_B[I]	:= GVL_1.DATA_RB_B.MAX_ACC;
	JERK_B[I]	:= GVL_1.DATA_RB_B.MAX_JERK;
	TORQUE_B[I]	:= GVL_1.DATA_RB_B.MAX_TOQUE;
END_FOR;
SMC_GroupSetAxisLimitFactors_A( AxisGroup 		:= SCARA_A, Execute := TRUE,
								VelFactors		:= VEL_A,
								AccFactors		:= ACC_A,
								JerkFactors		:= JERK_A,
								TorqueFactors	:= TORQUE_A,
								Done	=>,
								Busy	=>,
								Error	=>,
								ErrorID	=>);
SMC_GroupSetAxisLimitFactors_B( AxisGroup 		:= SCARA_B, Execute := TRUE,
								VelFactors		:= VEL_B,
								AccFactors		:= ACC_B,
								JerkFactors		:= JERK_B,
								TorqueFactors	:= TORQUE_B,
								Done	=>,
								Busy	=>,
								Error	=>,
								ErrorID	=>);
GVL.HMI_MAIN.Enable_Dynamics_Limit := FALSE;	
END_WHILE;
END_ACTION

END_PROGRAM

// Just_Motion_Control_x86_64_Linux_SM_WV/Application/PRG_ROBOT/POU_COORDINATE_
PROGRAM POU_COORDINATE_
VAR
	SMC_GroupSetTool_RBA: SMC_GroupSetTool;
	SMC_GroupSetTool_RBb: SMC_GroupSetTool;
	
	Pos_ORG				    : SM3_Robotics.MC_COORD_REF := (X:= 0, Y:= 0, Z:= 0, a := 0,B := 0, C:= 0);
	Point_offsetool_RBA		: SM3_Robotics.MC_COORD_REF := (X:= 0, Y:= 0, Z:= 0, a := 0, C:= 0);
	Point_offsetool_RBB		: SM3_Robotics.MC_COORD_REF := (X:= 0, Y:= 0, Z:= 0, a := 0);
	
	MC_SetCoordinateTransform_rba: MC_SetCoordinateTransform ;
	Coor_trans_RBA: SM3_Robotics.MC_COORD_REF := (X:= 0, Y:= 0, Z:= 0, a := 0,B := 0, C:= 0);
	MC_SetCoordinateTransform_rbb: MC_SetCoordinateTransform;
	Coor_trans_RBb: SM3_Robotics.MC_COORD_REF := (X:= 0, Y:= 0, Z:= 0, a := 0,B := 0, C:= 0);
	SMC_SetKinConfiguration_rba: SMC_SetKinConfiguration;	

	pre_Select_Tool_A, pre_Select_Tool_B : WORD;

	Convert_A_MCS, Convert_A_WCS, Convert_A_PCS_1,Convert_A_PCS_2, Convert_A_TCS_1, Convert_A_TCS_2,
	Convert_A_TCS_3, Convert_A_TCS_4, Convert_A_TCS_5  : SMC_GroupConvertPosition;
	Convert_B_MCS, Convert_B_WCS, Convert_B_PCS_1,Convert_B_PCS_2, Convert_B_TCS_1, Convert_B_TCS_2,
	Convert_B_TCS_3, Convert_B_TCS_4, Convert_B_TCS_5  : SMC_GroupConvertPosition;
	
	Pos_In: SM3_Robotics.SMC_POS_REF;
	Coor_trans_A: SM3_Robotics.SMC_COORD_SYSTEM;
	
	Tool_A_1, Tool_A_2, Tool_A_3, Tool_A_4, Tool_A_5,
	Tool_B_1, Tool_B_2, Tool_B_3, Tool_B_4, Tool_B_5	 : SM3_Robotics.MC_COORD_REF;
	
	Pos_Out_A_MCS, Pos_Out_A_WCS, Pos_Out_A_PCS_1, Pos_Out_A_PCS_2, Pos_Out_A_TCS_1, Pos_Out_A_TCS_2, Pos_Out_A_TCS_3, Pos_Out_A_TCS_4, Pos_Out_A_TCS_5,
	Pos_Out_B_MCS, Pos_Out_B_WCS, Pos_Out_B_PCS_1, Pos_Out_B_PCS_2, Pos_Out_B_TCS_1, Pos_Out_B_TCS_2, Pos_Out_B_TCS_3, Pos_Out_B_TCS_4, Pos_Out_B_TCS_5  : SM3_Robotics.SMC_POS_REF;
	
	CONFIG_: SM3_Robotics.TRAFO.CONFIGDATA;

END_VAR

VAR
	udiLastToolApplyRequestA : UDINT := 0;
	xSetToolExecuteA : BOOL := FALSE;
	udiLastToolApplyRequestB : UDINT;
	xSetToolExecuteB : BOOL;
	 
END_VAR

ACT_LOGIC();
ACT_CFC();
ACT_Conver_Pos();

ACTION ACT_CFC:
Convert_B_TCS_2(
    AxisGroup := SCARA_B,
    PositionIn := POU_MONITOR_ROBOT.RB2_POS_ACS,
    Enable := TRUE,
    CoordSystemIn := 0,
    CoordSystemOut := 1,
    UseToolOffsetParameter := TRUE,
    ToolOffset := Tool_B_2); // SMC_GroupConvertPosition
Convert_A_PCS_2(
    AxisGroup := SCARA_A,
    PositionIn := POU_MONITOR_ROBOT.RB1_POS_ACS,
    Enable := TRUE,
    CoordSystemIn := 0,
    CoordSystemOut := 4,
    UseToolOffsetParameter := TRUE,
    ToolOffset := Pos_ORG); // SMC_GroupConvertPosition
Convert_A_PCS_2(
    AxisGroup := SCARA_A,
    PositionIn := POU_MONITOR_ROBOT.RB2_POS_ACS,
    Enable := TRUE,
    CoordSystemIn := 0,
    CoordSystemOut := 4,
    UseToolOffsetParameter := TRUE,
    ToolOffset := Pos_ORG); // SMC_GroupConvertPosition
Convert_A_TCS_5(
    AxisGroup := SCARA_A,
    PositionIn := POU_MONITOR_ROBOT.RB1_POS_ACS,
    Enable := TRUE,
    CoordSystemIn := 0,
    CoordSystemOut := 1,
    UseToolOffsetParameter := TRUE,
    ToolOffset := Tool_A_5); // SMC_GroupConvertPosition
Pos_Out_B_TCS_2 := Convert_B_TCS_2.PositionOut;
Convert_A_WCS(
    AxisGroup := SCARA_A,
    PositionIn := POU_MONITOR_ROBOT.RB1_POS_ACS,
    Enable := TRUE,
    CoordSystemIn := 0,
    CoordSystemOut := 2,
    UseToolOffsetParameter := TRUE,
    ToolOffset := Pos_ORG); // SMC_GroupConvertPosition
MC_SetCoordinateTransform_rba(
    AxisGroup := SCARA_A,
    Execute := GVL.RB_A.HOME,
    CoordTransform := Coor_trans_RBA,
    CoordSystem := GVL.RB_A.COORD); // MC_SetCoordinateTransform
Convert_B_TCS_1(
    AxisGroup := SCARA_B,
    PositionIn := POU_MONITOR_ROBOT.RB2_POS_ACS,
    Enable := TRUE,
    CoordSystemIn := 0,
    CoordSystemOut := 1,
    UseToolOffsetParameter := TRUE,
    ToolOffset := Tool_B_1); // SMC_GroupConvertPosition
Convert_A_PCS_1(
    AxisGroup := SCARA_A,
    PositionIn := POU_MONITOR_ROBOT.RB1_POS_ACS,
    Enable := TRUE,
    CoordSystemIn := 0,
    CoordSystemOut := 3,
    UseToolOffsetParameter := TRUE,
    ToolOffset := Pos_ORG); // SMC_GroupConvertPosition
SMC_GroupSetTool_RBA(AxisGroup := SCARA_A, Execute := xSetToolExecuteA, ToolOffset := Point_offsetool_RBA); // SMC_GroupSetTool
Pos_Out_A_PCS_2 := Convert_A_PCS_2.PositionOut;
Convert_B_WCS(
    AxisGroup := SCARA_B,
    PositionIn := POU_MONITOR_ROBOT.RB2_POS_ACS,
    Enable := TRUE,
    CoordSystemIn := 0,
    CoordSystemOut := 2,
    UseToolOffsetParameter := TRUE,
    ToolOffset := Pos_ORG); // SMC_GroupConvertPosition
Convert_A_TCS_4(
    AxisGroup := SCARA_A,
    PositionIn := POU_MONITOR_ROBOT.RB1_POS_ACS,
    Enable := TRUE,
    CoordSystemIn := 0,
    CoordSystemOut := 1,
    UseToolOffsetParameter := TRUE,
    ToolOffset := Tool_A_4); // SMC_GroupConvertPosition
Pos_Out_B_TCS_1 := Convert_B_TCS_1.PositionOut;
Convert_B_TCS_5(
    AxisGroup := SCARA_B,
    PositionIn := POU_MONITOR_ROBOT.RB2_POS_ACS,
    Enable := TRUE,
    CoordSystemIn := 0,
    CoordSystemOut := 1,
    UseToolOffsetParameter := TRUE,
    ToolOffset := Tool_B_5); // SMC_GroupConvertPosition
Convert_A_TCS_3(
    AxisGroup := SCARA_A,
    PositionIn := POU_MONITOR_ROBOT.RB1_POS_ACS,
    Enable := TRUE,
    CoordSystemIn := 0,
    CoordSystemOut := 1,
    UseToolOffsetParameter := TRUE,
    ToolOffset := Tool_A_3); // SMC_GroupConvertPosition
Pos_Out_B_PCS_2 := Convert_A_PCS_2.PositionOut;
Pos_Out_A_TCS_5 := Convert_A_TCS_5.PositionOut;
MC_SetCoordinateTransform_rbb(
    AxisGroup := SCARA_B,
    Execute := GVL.RB_B.HOME,
    CoordTransform := Coor_trans_RBb,
    CoordSystem := GVL.RB_B.COORD); // MC_SetCoordinateTransform
Pos_Out_A_PCS_1 := Convert_A_PCS_1.PositionOut;
Convert_B_MCS(
    AxisGroup := SCARA_B,
    PositionIn := POU_MONITOR_ROBOT.RB2_POS_ACS,
    Enable := TRUE,
    CoordSystemIn := 0,
    CoordSystemOut := 1,
    UseToolOffsetParameter := TRUE,
    ToolOffset := Pos_ORG); // SMC_GroupConvertPosition
Pos_Out_B_MCS := Convert_B_MCS.PositionOut;
SMC_GroupSetTool_RBb(AxisGroup := SCARA_B, Execute := xSetToolExecuteB, ToolOffset := Point_offsetool_RBB); // SMC_GroupSetTool
Pos_Out_A_WCS := Convert_A_WCS.PositionOut;
Pos_Out_B_WCS := Convert_B_WCS.PositionOut;
Convert_B_TCS_4(
    AxisGroup := SCARA_A,
    PositionIn := POU_MONITOR_ROBOT.RB2_POS_ACS,
    Enable := TRUE,
    CoordSystemIn := 0,
    CoordSystemOut := 1,
    UseToolOffsetParameter := TRUE,
    ToolOffset := Tool_B_4); // SMC_GroupConvertPosition
Pos_Out_B_TCS_4 := Convert_B_TCS_4.PositionOut;
Convert_A_TCS_2(
    AxisGroup := SCARA_A,
    PositionIn := POU_MONITOR_ROBOT.RB1_POS_ACS,
    Enable := TRUE,
    CoordSystemIn := 0,
    CoordSystemOut := 1,
    UseToolOffsetParameter := TRUE,
    ToolOffset := Tool_A_2); // SMC_GroupConvertPosition
Pos_Out_A_TCS_2 := Convert_A_TCS_2.PositionOut;
Pos_Out_A_TCS_4 := Convert_A_TCS_4.PositionOut;
Pos_Out_B_TCS_5 := Convert_B_TCS_5.PositionOut;
Convert_B_TCS_3(
    AxisGroup := SCARA_B,
    PositionIn := POU_MONITOR_ROBOT.RB2_POS_ACS,
    Enable := TRUE,
    CoordSystemIn := 0,
    CoordSystemOut := 1,
    UseToolOffsetParameter := TRUE,
    ToolOffset := Tool_B_3); // SMC_GroupConvertPosition
Pos_Out_B_TCS_3 := Convert_B_TCS_3.PositionOut;
Convert_A_TCS_1(
    AxisGroup := SCARA_A,
    PositionIn := POU_MONITOR_ROBOT.RB1_POS_ACS,
    Enable := TRUE,
    CoordSystemIn := 0,
    CoordSystemOut := 1,
    UseToolOffsetParameter := TRUE,
    ToolOffset := Tool_A_1); // SMC_GroupConvertPosition
Pos_Out_A_TCS_1 := Convert_A_TCS_1.PositionOut;
Pos_Out_A_TCS_3 := Convert_A_TCS_3.PositionOut;
Convert_B_PCS_1(
    AxisGroup := SCARA_B,
    PositionIn := POU_MONITOR_ROBOT.RB1_POS_ACS,
    Enable := TRUE,
    CoordSystemIn := 0,
    CoordSystemOut := 3,
    UseToolOffsetParameter := TRUE,
    ToolOffset := Pos_ORG); // SMC_GroupConvertPosition
Pos_Out_A_PCS_1 := Convert_B_PCS_1.PositionOut;
Convert_A_MCS(
    AxisGroup := SCARA_A,
    PositionIn := POU_MONITOR_ROBOT.RB1_POS_ACS,
    Enable := TRUE,
    CoordSystemIn := 0,
    CoordSystemOut := 1,
    UseToolOffsetParameter := TRUE,
    ToolOffset := Pos_ORG); // SMC_GroupConvertPosition
Pos_Out_A_MCS := Convert_A_MCS.PositionOut;
END_ACTION

ACTION ACT_Conver_Pos:
{region "1. CONVERT_A"}
// ACS
GVL.COOR_A_CONVERT[0].X := TO_REAL(POU_MONITOR_ROBOT.RB1_POS_ACS.a.a0);
GVL.COOR_A_CONVERT[0].Y := TO_REAL(POU_MONITOR_ROBOT.RB1_POS_ACS.a.a1);
GVL.COOR_A_CONVERT[0].Z := TO_REAL(POU_MONITOR_ROBOT.RB1_POS_ACS.a.a2);
GVL.COOR_A_CONVERT[0].A := TO_REAL(POU_MONITOR_ROBOT.RB1_POS_ACS.a.a3);	
GVL.COOR_A_CONVERT[0].B := TO_REAL(POU_MONITOR_ROBOT.RB1_POS_ACS.a.a4);
GVL.COOR_A_CONVERT[0].C := TO_REAL(POU_MONITOR_ROBOT.RB1_POS_ACS.a.a5); 
// MCS
GVL.COOR_A_CONVERT[1].X := TO_REAL(Pos_Out_A_MCS.c.X);
GVL.COOR_A_CONVERT[1].Y := TO_REAL(Pos_Out_A_MCS.c.Y);
GVL.COOR_A_CONVERT[1].Z := TO_REAL(Pos_Out_A_MCS.c.Z);
GVL.COOR_A_CONVERT[1].A := TO_REAL(Pos_Out_A_MCS.c.A);	
GVL.COOR_A_CONVERT[1].B := TO_REAL(Pos_Out_A_MCS.c.B);
GVL.COOR_A_CONVERT[1].C := TO_REAL(Pos_Out_A_MCS.c.C); 
// WCS
GVL.COOR_A_CONVERT[2].X := TO_REAL(Pos_Out_A_WCS.c.X);
GVL.COOR_A_CONVERT[2].Y := TO_REAL(Pos_Out_A_WCS.c.Y);
GVL.COOR_A_CONVERT[2].Z := TO_REAL(Pos_Out_A_WCS.c.Z);
GVL.COOR_A_CONVERT[2].A := TO_REAL(Pos_Out_A_WCS.c.A);	
GVL.COOR_A_CONVERT[2].B := TO_REAL(Pos_Out_A_WCS.c.B);
GVL.COOR_A_CONVERT[2].C := TO_REAL(Pos_Out_A_WCS.c.C); 
// PCS_1
GVL.COOR_A_CONVERT[3].X := TO_REAL(Pos_Out_A_PCS_1.c.X);
GVL.COOR_A_CONVERT[3].Y := TO_REAL(Pos_Out_A_PCS_1.c.Y);
GVL.COOR_A_CONVERT[3].Z := TO_REAL(Pos_Out_A_PCS_1.c.Z);
GVL.COOR_A_CONVERT[3].A := TO_REAL(Pos_Out_A_PCS_1.c.A);	
GVL.COOR_A_CONVERT[3].B := TO_REAL(Pos_Out_A_PCS_1.c.B);
GVL.COOR_A_CONVERT[3].C := TO_REAL(Pos_Out_A_PCS_1.c.C); 
// PCS_2
GVL.COOR_A_CONVERT[4].X := TO_REAL(Pos_Out_A_PCS_2.c.X);
GVL.COOR_A_CONVERT[4].Y := TO_REAL(Pos_Out_A_PCS_2.c.Y);
GVL.COOR_A_CONVERT[4].Z := TO_REAL(Pos_Out_A_PCS_2.c.Z);
GVL.COOR_A_CONVERT[4].A := TO_REAL(Pos_Out_A_PCS_2.c.A);	
GVL.COOR_A_CONVERT[4].B := TO_REAL(Pos_Out_A_PCS_2.c.B);
GVL.COOR_A_CONVERT[4].C := TO_REAL(Pos_Out_A_PCS_2.c.C);	
// TCS_1
GVL.COOR_A_CONVERT[5].X := TO_REAL(Pos_Out_A_TCS_1.c.X);
GVL.COOR_A_CONVERT[5].Y := TO_REAL(Pos_Out_A_TCS_1.c.Y);
GVL.COOR_A_CONVERT[5].Z := TO_REAL(Pos_Out_A_TCS_1.c.Z);
GVL.COOR_A_CONVERT[5].A := TO_REAL(Pos_Out_A_TCS_1.c.A);	
GVL.COOR_A_CONVERT[5].B := TO_REAL(Pos_Out_A_TCS_1.c.B);
GVL.COOR_A_CONVERT[5].C := TO_REAL(Pos_Out_A_TCS_1.c.C);
// TCS_2
GVL.COOR_A_CONVERT[6].X := TO_REAL(Pos_Out_A_TCS_2.c.X);
GVL.COOR_A_CONVERT[6].Y := TO_REAL(Pos_Out_A_TCS_2.c.Y);
GVL.COOR_A_CONVERT[6].Z := TO_REAL(Pos_Out_A_TCS_2.c.Z);
GVL.COOR_A_CONVERT[6].A := TO_REAL(Pos_Out_A_TCS_2.c.A);	
GVL.COOR_A_CONVERT[6].B := TO_REAL(Pos_Out_A_TCS_2.c.B);
GVL.COOR_A_CONVERT[6].C := TO_REAL(Pos_Out_A_TCS_2.c.C);		 
{endregion}

{region "2. CONVERT_B"}
// ACS
GVL.COOR_B_CONVERT[0].X := TO_REAL(POU_MONITOR_ROBOT.RB2_POS_ACS.a.a0);
GVL.COOR_B_CONVERT[0].Y := TO_REAL(POU_MONITOR_ROBOT.RB2_POS_ACS.a.a1);
GVL.COOR_B_CONVERT[0].Z := TO_REAL(POU_MONITOR_ROBOT.RB2_POS_ACS.a.a2);
GVL.COOR_B_CONVERT[0].A := TO_REAL(POU_MONITOR_ROBOT.RB2_POS_ACS.a.a3);	
GVL.COOR_B_CONVERT[0].B := TO_REAL(POU_MONITOR_ROBOT.RB2_POS_ACS.a.a4);
GVL.COOR_B_CONVERT[0].C := TO_REAL(POU_MONITOR_ROBOT.RB2_POS_ACS.a.a5); 
// MCS
GVL.COOR_B_CONVERT[1].X := TO_REAL(Pos_Out_B_MCS.c.X);
GVL.COOR_B_CONVERT[1].Y := TO_REAL(Pos_Out_B_MCS.c.Y);
GVL.COOR_B_CONVERT[1].Z := TO_REAL(Pos_Out_B_MCS.c.Z);
GVL.COOR_B_CONVERT[1].A := TO_REAL(Pos_Out_B_MCS.c.A);	
GVL.COOR_B_CONVERT[1].B := TO_REAL(Pos_Out_B_MCS.c.B);
GVL.COOR_B_CONVERT[1].C := TO_REAL(Pos_Out_B_MCS.c.C); 
// WCS
GVL.COOR_B_CONVERT[2].X := TO_REAL(Pos_Out_B_WCS.c.X);
GVL.COOR_B_CONVERT[2].Y := TO_REAL(Pos_Out_B_WCS.c.Y);
GVL.COOR_B_CONVERT[2].Z := TO_REAL(Pos_Out_B_WCS.c.Z);
GVL.COOR_B_CONVERT[2].A := TO_REAL(Pos_Out_B_WCS.c.A);	
GVL.COOR_B_CONVERT[2].B := TO_REAL(Pos_Out_B_WCS.c.B);
GVL.COOR_B_CONVERT[2].C := TO_REAL(Pos_Out_B_WCS.c.C); 
// PCS_1
GVL.COOR_B_CONVERT[3].X := TO_REAL(Pos_Out_B_PCS_1.c.X);
GVL.COOR_B_CONVERT[3].Y := TO_REAL(Pos_Out_B_PCS_1.c.Y);
GVL.COOR_B_CONVERT[3].Z := TO_REAL(Pos_Out_B_PCS_1.c.Z);
GVL.COOR_B_CONVERT[3].A := TO_REAL(Pos_Out_B_PCS_1.c.A);	
GVL.COOR_B_CONVERT[3].B := TO_REAL(Pos_Out_B_PCS_1.c.B);
GVL.COOR_B_CONVERT[3].C := TO_REAL(Pos_Out_B_PCS_1.c.C); 
// PCS_2
GVL.COOR_B_CONVERT[4].X := TO_REAL(Pos_Out_B_PCS_2.c.X);
GVL.COOR_B_CONVERT[4].Y := TO_REAL(Pos_Out_B_PCS_2.c.Y);
GVL.COOR_B_CONVERT[4].Z := TO_REAL(Pos_Out_B_PCS_2.c.Z);
GVL.COOR_B_CONVERT[4].A := TO_REAL(Pos_Out_B_PCS_2.c.A);	
GVL.COOR_B_CONVERT[4].B := TO_REAL(Pos_Out_B_PCS_2.c.B);
GVL.COOR_B_CONVERT[4].C := TO_REAL(Pos_Out_B_PCS_2.c.C);	
// TCS_1
GVL.COOR_B_CONVERT[5].X := TO_REAL(Pos_Out_B_TCS_1.c.X);
GVL.COOR_B_CONVERT[5].Y := TO_REAL(Pos_Out_B_TCS_1.c.Y);
GVL.COOR_B_CONVERT[5].Z := TO_REAL(Pos_Out_B_TCS_1.c.Z);
GVL.COOR_B_CONVERT[5].A := TO_REAL(Pos_Out_B_TCS_1.c.A);	
GVL.COOR_B_CONVERT[5].B := TO_REAL(Pos_Out_B_TCS_1.c.B);
GVL.COOR_B_CONVERT[5].C := TO_REAL(Pos_Out_B_TCS_1.c.C);
// TCS_2
GVL.COOR_B_CONVERT[6].X := TO_REAL(Pos_Out_B_TCS_2.c.X);
GVL.COOR_B_CONVERT[6].Y := TO_REAL(Pos_Out_B_TCS_2.c.Y);
GVL.COOR_B_CONVERT[6].Z := TO_REAL(Pos_Out_B_TCS_2.c.Z);
GVL.COOR_B_CONVERT[6].A := TO_REAL(Pos_Out_B_TCS_2.c.A);	
GVL.COOR_B_CONVERT[6].B := TO_REAL(Pos_Out_B_TCS_2.c.B);
GVL.COOR_B_CONVERT[6].C := TO_REAL(Pos_Out_B_TCS_2.c.C);		 
{endregion}
END_ACTION

ACTION ACT_LOGIC:
{region "1. Select_Tool"}
/// ROBOT A
	 
//=============================================================================
// ROBOT A - SELECT / APPLY TOOL TCP
//-----------------------------------------------------------------------------
// Quy ước:
// Number_Tool = 0 : Không sử dụng Tool Offset.
// Number_Tool = 1 : Tool 1.
// Number_Tool = 2 : Tool 2.
// ...
//
// Nguồn TCP duy nhất:
// GVL.g_aToolConfigA[ToolID].ToolTCP
//
// Tool được Apply lại khi:
// 1. Number_Tool thay đổi.
// 2. Có ApplyRequest mới, kể cả Number_Tool không đổi.
//
// SMC_GroupSetTool_RBA đã được đặt sẵn trên FBD.
// Chân Execute của SMC_GroupSetTool_RBA phải nối với xSetToolExecuteA.
//=============================================================================

GVL.g_xRobotAToolApplyDone := FALSE;


//=============================================================================
// 01. PHÁT HIỆN YÊU CẦU APPLY TOOL MỚI
//=============================================================================
IF ((pre_Select_Tool_A <> GVL.RB_A.Number_Tool)
OR (GVL.g_udiRobotAToolApplyRequestA <> udiLastToolApplyRequestA))
AND NOT xSetToolExecuteA THEN

    //---------------------------------------------------------------------
    // Xóa trạng thái transaction trước.
    //---------------------------------------------------------------------
    GVL.g_xRobotAToolApplyBusy := TRUE;
    GVL.g_xRobotAToolApplyDone := FALSE;
    GVL.g_xRobotAToolApplyError := FALSE;
    GVL.g_udiRobotAToolApplyErrorID := 0;


    //---------------------------------------------------------------------
    // TOOL 0 - KHÔNG SỬ DỤNG TOOL OFFSET
    //---------------------------------------------------------------------
    IF GVL.RB_A.Number_Tool = 0 THEN

        Point_offsetool_RBA := Pos_ORG;


    //---------------------------------------------------------------------
    // TOOL 1..C_MAX_TOOLS
    //---------------------------------------------------------------------
    ELSIF GVL.RB_A.Number_Tool >= 1
    AND GVL.RB_A.Number_Tool <= GVL.C_MAX_TOOLS THEN

        // Lấy trực tiếp TCP của Tool đang được chọn.
        Point_offsetool_RBA.X := TO_LREAL(GVL.g_aToolConfigA[GVL.RB_A.Number_Tool].ToolTCP.X);
        Point_offsetool_RBA.Y := TO_LREAL(GVL.g_aToolConfigA[GVL.RB_A.Number_Tool].ToolTCP.Y);
        Point_offsetool_RBA.Z := TO_LREAL(GVL.g_aToolConfigA[GVL.RB_A.Number_Tool].ToolTCP.Z);
        Point_offsetool_RBA.A := TO_LREAL(GVL.g_aToolConfigA[GVL.RB_A.Number_Tool].ToolTCP.A);
        Point_offsetool_RBA.B := TO_LREAL(0);
        Point_offsetool_RBA.C := TO_LREAL(0);


    //---------------------------------------------------------------------
    // TOOL NUMBER KHÔNG HỢP LỆ
    //---------------------------------------------------------------------
    ELSE

        GVL.g_xRobotAToolApplyBusy := FALSE;
        GVL.g_xRobotAToolApplyDone := FALSE;
        GVL.g_xRobotAToolApplyError := TRUE;

        // Lỗi nội bộ: Number_Tool ngoài phạm vi cho phép.
        GVL.g_udiRobotAToolApplyErrorID := 10001;

    END_IF;


    //---------------------------------------------------------------------
    // Chỉ phát Execute nếu Tool Number hợp lệ.
    //---------------------------------------------------------------------
    IF NOT GVL.g_xRobotAToolApplyError THEN

        // Ghi nhớ Tool đang Apply.
        pre_Select_Tool_A := GVL.RB_A.Number_Tool;

        // Ghi nhớ Request đang xử lý.
        udiLastToolApplyRequestA := GVL.g_udiRobotAToolApplyRequestA;

        // Phát Execute cho SMC_GroupSetTool_RBA trên FBD.
        xSetToolExecuteA := TRUE;

    END_IF;

END_IF;


//=============================================================================
// 02. SMC_GroupSetTool HOÀN THÀNH
//-----------------------------------------------------------------------------
// SMC_GroupSetTool_RBA được gọi trên FBD.
// Ở đây chỉ đọc Done / Error của instance đó.
//=============================================================================
IF xSetToolExecuteA AND SMC_GroupSetTool_RBA.Done THEN

    // Hạ Execute để tạo cạnh mới cho lần Apply tiếp theo.
    xSetToolExecuteA := FALSE;

    // Transaction hoàn thành.
    GVL.g_xRobotAToolApplyBusy := FALSE;
    GVL.g_xRobotAToolApplyDone := TRUE;
    GVL.g_xRobotAToolApplyError := FALSE;
    GVL.g_udiRobotAToolApplyErrorID := 0;

    // Xác nhận đúng Request đã được Apply.
    GVL.g_udiRobotAToolAppliedRequestA := udiLastToolApplyRequestA;

END_IF;


//=============================================================================
// 03. SMC_GroupSetTool ERROR
//=============================================================================
IF xSetToolExecuteA AND SMC_GroupSetTool_RBA.Error THEN

    // Kết thúc transaction hiện tại.
    xSetToolExecuteA := FALSE;

    GVL.g_xRobotAToolApplyBusy := FALSE;
    GVL.g_xRobotAToolApplyDone := FALSE;
    GVL.g_xRobotAToolApplyError := TRUE;

    // Chuyển ErrorID của SoftMotion ra hệ thống chung.
    GVL.g_udiRobotAToolApplyErrorID := TO_UDINT(SMC_GroupSetTool_RBA.ErrorID);

END_IF;
	 
		  
			   
// IF pre_Select_Tool_A <> GVL.RB_A.Number_Tool THEN
// 
// CASE GVL.RB_A.Number_Tool OF
// 	0: 	
// 		Point_offsetool_RBA := Pos_ORG;
// 
// 	1:  
// 		Point_offsetool_RBA.X := TO_LREAL(GVL_2.A_Tool[0].X);
// 		Point_offsetool_RBA.Y := TO_LREAL(GVL_2.A_Tool[0].Y);
// 		Point_offsetool_RBA.Z := TO_LREAL(GVL_2.A_Tool[0].Z);
// 		Point_offsetool_RBA.A := TO_LREAL(GVL_2.A_Tool[0].A);
// 		Point_offsetool_RBA.B := TO_LREAL(GVL_2.A_Tool[0].B);
// 		Point_offsetool_RBA.C := TO_LREAL(GVL_2.A_Tool[0].C);
// 		
// 	2:  
// 		Point_offsetool_RBA.X := TO_LREAL(GVL_2.A_Tool[1].X);
// 		Point_offsetool_RBA.Y := TO_LREAL(GVL_2.A_Tool[1].Y);
// 		Point_offsetool_RBA.Z := TO_LREAL(GVL_2.A_Tool[1].Z);
// 		Point_offsetool_RBA.A := TO_LREAL(GVL_2.A_Tool[1].A);
// 		Point_offsetool_RBA.B := TO_LREAL(GVL_2.A_Tool[1].B);
// 		Point_offsetool_RBA.C := TO_LREAL(GVL_2.A_Tool[1].C);
// 	
// 	3:  
// 		Point_offsetool_RBA.X := TO_LREAL(GVL_2.A_Tool[2].X);
// 		Point_offsetool_RBA.Y := TO_LREAL(GVL_2.A_Tool[2].Y);
// 		Point_offsetool_RBA.Z := TO_LREAL(GVL_2.A_Tool[2].Z);
// 		Point_offsetool_RBA.A := TO_LREAL(GVL_2.A_Tool[2].A);
// 		Point_offsetool_RBA.B := TO_LREAL(GVL_2.A_Tool[2].B);
// 		Point_offsetool_RBA.C := TO_LREAL(GVL_2.A_Tool[2].C);
// 	4:  
// 		Point_offsetool_RBA.X := TO_LREAL(GVL_2.A_Tool[3].X);
// 		Point_offsetool_RBA.Y := TO_LREAL(GVL_2.A_Tool[3].Y);
// 		Point_offsetool_RBA.Z := TO_LREAL(GVL_2.A_Tool[3].Z);
// 		Point_offsetool_RBA.A := TO_LREAL(GVL_2.A_Tool[3].A);
// 		Point_offsetool_RBA.B := TO_LREAL(GVL_2.A_Tool[3].B);
// 		Point_offsetool_RBA.C := TO_LREAL(GVL_2.A_Tool[3].C);
// 	5:  
// 		Point_offsetool_RBA.X := TO_LREAL(GVL_2.A_Tool[4].X);
// 		Point_offsetool_RBA.Y := TO_LREAL(GVL_2.A_Tool[4].Y);
// 		Point_offsetool_RBA.Z := TO_LREAL(GVL_2.A_Tool[4].Z);
// 		Point_offsetool_RBA.A := TO_LREAL(GVL_2.A_Tool[4].A);
// 		Point_offsetool_RBA.B := TO_LREAL(GVL_2.A_Tool[4].B);
// 		Point_offsetool_RBA.C := TO_LREAL(GVL_2.A_Tool[4].C);			 
// END_CASE	
// 	 SMC_GroupSetTool_RBA.Execute := TRUE;
// ELSE
// 	SMC_GroupSetTool_RBA.Execute := FALSE;
// END_IF
// pre_Select_Tool_A := GVL.RB_A.Number_Tool;
	 
		  
			   
					
// POU_COORDINATE_ - ROBOT B TOOL APPLY
// Thêm local: udiLastToolApplyRequestB : UDINT; xSetToolExecuteB : BOOL;
// Thay phần Robot B để dùng g_aToolConfigB và handshake B riêng.
// Chân Execute của SMC_GroupSetTool_RBb phải nối xSetToolExecuteB.

GVL.g_xRobotBToolApplyDone := FALSE;

IF ((pre_Select_Tool_B <> GVL.RB_B.Number_Tool) OR (GVL.g_udiRobotBToolApplyRequestB <> udiLastToolApplyRequestB))
AND NOT xSetToolExecuteB THEN
    GVL.g_xRobotBToolApplyBusy := TRUE;
    GVL.g_xRobotBToolApplyDone := FALSE;
    GVL.g_xRobotBToolApplyError := FALSE;
    GVL.g_udiRobotBToolApplyErrorID := 0;

    IF GVL.RB_B.Number_Tool = 0 THEN
        Point_offsetool_RBB := Pos_ORG;
    ELSIF GVL.RB_B.Number_Tool >= 1 AND GVL.RB_B.Number_Tool <= GVL.C_MAX_TOOLS THEN
        Point_offsetool_RBB.X := TO_LREAL(GVL.g_aToolConfigB[GVL.RB_B.Number_Tool].ToolTCP.X);
        Point_offsetool_RBB.Y := TO_LREAL(GVL.g_aToolConfigB[GVL.RB_B.Number_Tool].ToolTCP.Y);
        Point_offsetool_RBB.Z := TO_LREAL(GVL.g_aToolConfigB[GVL.RB_B.Number_Tool].ToolTCP.Z);
        Point_offsetool_RBB.A := TO_LREAL(GVL.g_aToolConfigB[GVL.RB_B.Number_Tool].ToolTCP.A);
        Point_offsetool_RBB.B := 0.0;
        Point_offsetool_RBB.C := 0.0;
        pre_Select_Tool_B := GVL.RB_B.Number_Tool;
        udiLastToolApplyRequestB := GVL.g_udiRobotBToolApplyRequestB;
        xSetToolExecuteB := TRUE;
    ELSE
        GVL.g_xRobotBToolApplyBusy := FALSE;
        GVL.g_xRobotBToolApplyError := TRUE;
        GVL.g_udiRobotBToolApplyErrorID := 10001;
    END_IF;
END_IF;

IF xSetToolExecuteB AND SMC_GroupSetTool_RBb.Done THEN
    xSetToolExecuteB := FALSE;
    GVL.g_xRobotBToolApplyBusy := FALSE;
    GVL.g_xRobotBToolApplyDone := TRUE;
    GVL.g_udiRobotBToolAppliedRequestB := udiLastToolApplyRequestB;
END_IF;

IF xSetToolExecuteB AND SMC_GroupSetTool_RBb.Error THEN
    xSetToolExecuteB := FALSE;
    GVL.g_xRobotBToolApplyBusy := FALSE;
    GVL.g_xRobotBToolApplyError := TRUE;
    GVL.g_udiRobotBToolApplyErrorID := TO_UDINT(SMC_GroupSetTool_RBb.ErrorID);
END_IF;
						 
	 
// /// ROBOT B
// IF pre_Select_Tool_B <> GVL.RB_B.Number_Tool THEN
// 	
// CASE GVL.RB_b.Number_Tool OF
// 	0: 	
// 		Point_offsetool_RBB := Pos_ORG;
// 	1:  
// 		Point_offsetool_RBB.X := TO_LREAL(GVL_2.B_Tool[0].X);
// 		Point_offsetool_RBB.Y := TO_LREAL(GVL_2.B_Tool[0].Y);
// 		Point_offsetool_RBB.Z := TO_LREAL(GVL_2.B_Tool[0].Z);
// 		Point_offsetool_RBB.A := TO_LREAL(GVL_2.B_Tool[0].A);
// 		Point_offsetool_RBB.B := TO_LREAL(GVL_2.B_Tool[0].B);
// 		Point_offsetool_RBB.C := TO_LREAL(GVL_2.B_Tool[0].C);		
// 	2:  
// 		Point_offsetool_RBB.X := TO_LREAL(GVL_2.B_Tool[1].X);
// 		Point_offsetool_RBB.Y := TO_LREAL(GVL_2.B_Tool[1].Y);
// 		Point_offsetool_RBB.Z := TO_LREAL(GVL_2.B_Tool[1].Z);
// 		Point_offsetool_RBB.A := TO_LREAL(GVL_2.B_Tool[1].A);
// 		Point_offsetool_RBB.B := TO_LREAL(GVL_2.B_Tool[1].B);
// 		Point_offsetool_RBB.C := TO_LREAL(GVL_2.B_Tool[1].C);
// 
// 	3:  
// 		Point_offsetool_RBB.X := TO_LREAL(GVL_2.B_Tool[2].X);
// 		Point_offsetool_RBB.Y := TO_LREAL(GVL_2.B_Tool[2].Y);
// 		Point_offsetool_RBB.Z := TO_LREAL(GVL_2.B_Tool[2].Z);
// 		Point_offsetool_RBB.A := TO_LREAL(GVL_2.B_Tool[2].A);
// 		Point_offsetool_RBB.B := TO_LREAL(GVL_2.B_Tool[2].B);
// 		Point_offsetool_RBB.C := TO_LREAL(GVL_2.B_Tool[2].C);
// 	4:  
// 		Point_offsetool_RBB.X := TO_LREAL(GVL_2.B_Tool[3].X);
// 		Point_offsetool_RBB.Y := TO_LREAL(GVL_2.B_Tool[3].Y);
// 		Point_offsetool_RBB.Z := TO_LREAL(GVL_2.B_Tool[3].Z);
// 		Point_offsetool_RBB.A := TO_LREAL(GVL_2.B_Tool[3].A);
// 		Point_offsetool_RBB.B := TO_LREAL(GVL_2.B_Tool[3].B);
// 		Point_offsetool_RBB.C := TO_LREAL(GVL_2.B_Tool[3].C);	
// 	5:  
// 		Point_offsetool_RBB.X := TO_LREAL(GVL_2.B_Tool[4].X);
// 		Point_offsetool_RBB.Y := TO_LREAL(GVL_2.B_Tool[4].Y);
// 		Point_offsetool_RBB.Z := TO_LREAL(GVL_2.B_Tool[4].Z);
// 		Point_offsetool_RBB.A := TO_LREAL(GVL_2.B_Tool[4].A);
// 		Point_offsetool_RBB.B := TO_LREAL(GVL_2.B_Tool[4].B);
// 		Point_offsetool_RBB.C := TO_LREAL(GVL_2.B_Tool[4].C);		 
// 
// END_CASE
// 	SMC_GroupSetTool_RBb.Execute := TRUE;
// ELSE
// 	SMC_GroupSetTool_RBb.Execute := FALSE;		
// END_IF
// pre_Select_Tool_B := GVL.RB_B.Number_Tool;
					
{endregion}
{region "2. SET COORDINATE SYSTEM"}	 
	Coor_trans_RBA.X := TO_LREAL(GVL_2.A_POS_COOR.X);
	Coor_trans_RBA.Y := TO_LREAL(GVL_2.A_POS_COOR.y);	 
	Coor_trans_RBA.Z := TO_LREAL(GVL_2.A_POS_COOR.z);
	Coor_trans_RBA.a := TO_LREAL(GVL_2.A_POS_COOR.A);
	Coor_trans_RBA.B := TO_LREAL(GVL_2.A_POS_COOR.b);	
	Coor_trans_RBA.C := TO_LREAL(GVL_2.A_POS_COOR.C);  
			   
	Coor_trans_RBb.X := TO_LREAL(GVL_2.B_POS_COOR.X);
	Coor_trans_RBb.Y := TO_LREAL(GVL_2.B_POS_COOR.y);	 
	Coor_trans_RBb.Z := TO_LREAL(GVL_2.B_POS_COOR.z);
	Coor_trans_RBb.a := TO_LREAL(GVL_2.B_POS_COOR.A);
	Coor_trans_RBb.B := TO_LREAL(GVL_2.B_POS_COOR.b);	
	Coor_trans_RBb.C := TO_LREAL(GVL_2.B_POS_COOR.C);  					

		  
{endregion}
	 
{region "3. Convert Pos___TOOL"}

	// TOOL_1
		Tool_A_1.X := TO_LREAL(GVL_2.A_Tool[0].X);
		Tool_A_1.Y := TO_LREAL(GVL_2.A_Tool[0].Y);
		Tool_A_1.Z := TO_LREAL(GVL_2.A_Tool[0].Z);
		Tool_A_1.A := TO_LREAL(GVL_2.A_Tool[0].A);
		Tool_A_1.B := TO_LREAL(GVL_2.A_Tool[0].B);
		Tool_A_1.C := TO_LREAL(GVL_2.A_Tool[0].C); 
	// TOOL_2
		Tool_A_2.X := TO_LREAL(GVL_2.A_Tool[1].X);
		Tool_A_2.Y := TO_LREAL(GVL_2.A_Tool[1].Y);
		Tool_A_2.Z := TO_LREAL(GVL_2.A_Tool[1].Z);
		Tool_A_2.A := TO_LREAL(GVL_2.A_Tool[1].A);
		Tool_A_2.B := TO_LREAL(GVL_2.A_Tool[1].B);
		Tool_A_2.C := TO_LREAL(GVL_2.A_Tool[1].C); 	


	// TOOL_1
		Tool_B_1.X := TO_LREAL(GVL_2.B_Tool[0].X);
		Tool_B_1.Y := TO_LREAL(GVL_2.B_Tool[0].Y);
		Tool_B_1.Z := TO_LREAL(GVL_2.B_Tool[0].Z);
		Tool_B_1.A := TO_LREAL(GVL_2.B_Tool[0].A);
		Tool_B_1.B := TO_LREAL(GVL_2.B_Tool[0].B);
		Tool_B_1.C := TO_LREAL(GVL_2.B_Tool[0].C); 
	// TOOL_2
		Tool_B_2.X := TO_LREAL(GVL_2.B_Tool[1].X);
		Tool_B_2.Y := TO_LREAL(GVL_2.B_Tool[1].Y);
		Tool_B_2.Z := TO_LREAL(GVL_2.B_Tool[1].Z);
		Tool_B_2.A := TO_LREAL(GVL_2.B_Tool[1].A);
		Tool_B_2.B := TO_LREAL(GVL_2.B_Tool[1].B);
		Tool_B_2.C := TO_LREAL(GVL_2.B_Tool[1].C); 
		
{endregion}
END_ACTION

END_PROGRAM

// Just_Motion_Control_x86_64_Linux_SM_WV/Application/FC_/F_CheckPositionReached
FUNCTION F_CheckPositionReached  : BOOL // Kiem tra toa do target va hien tai da chinh xac chua
VAR_INPUT
    Target, Actual : SMC_POS_REF;
    TolXYZ : LREAL;
    TolR   : LREAL;
END_VAR
VAR
END_VAR

F_CheckPositionReached :=
    (ABS(Target.c.X - Actual.c.X) <= TolXYZ) AND
    (ABS(Target.c.Y - Actual.c.Y) <= TolXYZ) AND
    (ABS(Target.c.Z - Actual.c.Z) <= TolXYZ) AND
	(ABS(Target.c.A - Actual.c.A) <= TolR) ;

END_FUNCTION

// Just_Motion_Control_x86_64_Linux_SM_WV/Application/FB_/FB_RunMoveL
FUNCTION_BLOCK FB_RunMoveL
VAR_INPUT
    Start       : BOOL;
    Item        : ST_MotionQueueItem;
    PositionIn  : SMC_POS_REF;
    CoordSystem : SMC_COORD_SYSTEM;

    AcceptTimeoutTime : TIME := T#2S;
    MoveTimeoutTime   : TIME := T#50S;
    PosCheckDelayTime : TIME := T#13MS;
END_VAR
VAR_IN_OUT
	AxisGroup   : AXIS_GROUP_REF_SM3;
END_VAR
VAR_OUTPUT
    Accepted       : BOOL;
    Done           : BOOL;
    Busy           : BOOL;
    Active         : BOOL;
    Error          : BOOL;
    Timeout        : BOOL;
    Aborted        : BOOL;
    ErrorID        : SMC_ERROR;
    ErrorID_Custom : INT;
    State          : E_MoveState;
END_VAR

VAR
	//--------------------------------------------------------
    // SoftMotion FB gốc
    //--------------------------------------------------------
    fbMoveL : MC_MoveLinearAbsolute;
	//--------------------------------------------------------
    // Timer
    //--------------------------------------------------------
    tAcceptTimeout : TON;
    tMoveTimeout   : TON;
    tPosCheckDelay : TON;

	//--------------------------------------------------------
    // Execute control
    //--------------------------------------------------------
    StartEdge    : BOOL;
    LastStart    : BOOL;
    ExecutePulse : BOOL;
	
	//--------------------------------------------------------
    // Target buffer
    //--------------------------------------------------------
    PosBuf : SMC_POS_REF;
	DonePosition : SM3_Robotics.SMC_POS_REF;

    //--------------------------------------------------------
    // Path dynamics
    //--------------------------------------------------------
    Vel  : LREAL;
    Acc  : LREAL;
    Dec  : LREAL;
    Jerk : LREAL;
	
	 //--------------------------------------------------------
    // Blending
    //--------------------------------------------------------
    BufferMode : SM3_Robotics.MC_BUFFER_MODE;
    TransMode  : SM3_Robotics.MC_TRANSITION_MODE;
    TransParam : ARRAY[0..(SMC_RCNST.MAX_TRANS_PARAMS - 1)] OF LREAL := [0.0, 0.0];
	//--------------------------------------------------------
    // Orientation
    //--------------------------------------------------------
    OrientationMode : SM3_Robotics.SMC_ORIENTATION_MODE;
	 //--------------------------------------------------------
    // Dynamic factors
    //--------------------------------------------------------
    VelFacLocal    : LREAL;
    AccFacLocal    : LREAL;
    JerkFacLocal   : LREAL;
    TorqueFacLocal : LREAL;
END_VAR

VAR CONSTANT
	C_BM_Buffered     : SM3_Robotics.MC_BUFFER_MODE := 1;
    C_BM_BlendingNext : SM3_Robotics.MC_BUFFER_MODE := 4;

    C_TM_CornerDistance : SM3_Robotics.MC_TRANSITION_MODE := 2;
    C_TM_None           : SM3_Robotics.MC_TRANSITION_MODE := 0;
    C_TM_StartVelocity  : SM3_Robotics.MC_TRANSITION_MODE := 1;
END_VAR

//============================================================
// FB_RunMoveL
//
// Chạy TCP theo đường thẳng tới PositionIn.
//
// Cơ chế giống FB_RunMoveP:
// - Giữ Execute đến CommandAccepted.
// - Accepted được latch.
// - Done được giữ để MotionManager đọc.
// - SkipPositionCheck dùng cho điểm bị ảnh hưởng blending.
//============================================================


//------------------------------------------------------------
// Phát hiện cạnh Start
//------------------------------------------------------------
StartEdge := Start AND NOT LastStart;
LastStart := Start;


//------------------------------------------------------------
// Execute mặc định FALSE.
// Chỉ bật ở MOVE_SEND / MOVE_WAIT_ACCEPT.
//------------------------------------------------------------
ExecutePulse := FALSE;


//============================================================
// STATE MACHINE
//============================================================
CASE State OF


    //========================================================
    // IDLE
    //========================================================
    E_MoveState.MOVE_IDLE:

        Accepted := FALSE;
        Done     := FALSE;
        Error    := FALSE;
        Timeout  := FALSE;
        Aborted  := FALSE;

        //Release := FALSE;

        ErrorID_Custom := 0;

        //----------------------------------------------------
        // Reset timer
        //----------------------------------------------------
        tAcceptTimeout(IN := FALSE);
        tMoveTimeout(IN := FALSE);
        tPosCheckDelay(IN := FALSE);


        //----------------------------------------------------
        // Chỉ nhận lệnh khi FB gốc đã rảnh
        //----------------------------------------------------
        IF Start
           AND NOT fbMoveL.Busy
           AND NOT fbMoveL.Active
        THEN

            //------------------------------------------------
            // Chốt tọa độ
            //------------------------------------------------
            PosBuf := PositionIn;


            //------------------------------------------------
            // SPEED
            //
            // Item.Speed > 0:
            //     speed riêng của step.
            //
            // Item.Speed <= 0:
            //     dùng speed hiện tại.
            //------------------------------------------------
            IF Item.Speed > 0.0 THEN
                Vel := Item.Speed;
            ELSE
				IF AxisGroup.m_id = SCARA_A.m_id THEN
                	Vel := GVL.A_CurrentMotionParam.Speed;
				ELSE
					Vel := GVL.B_CurrentMotionParam.Speed;
				END_IF
            END_IF;


            //------------------------------------------------
            // Dynamics hiện tại
            //------------------------------------------------

			IF AxisGroup.m_id = SCARA_A.m_id THEN
				IF Item.Acceleration > 0.0 THEN Acc := Item.Acceleration; ELSE Acc := GVL_1.DATA_RB_A.MOTION_ACC; END_IF;
				IF Item.Deceleration > 0.0 THEN Dec := Item.Deceleration; ELSE Dec := GVL_1.DATA_RB_A.MOTION_DEC; END_IF;
				IF Item.Jerk > 0.0 THEN Jerk := Item.Jerk; ELSE Jerk := GVL_1.DATA_RB_A.MOTION_JERK; END_IF;
			ELSE
				IF Item.Acceleration > 0.0 THEN Acc := Item.Acceleration; ELSE Acc := GVL_1.DATA_RB_B.MOTION_ACC; END_IF;
				IF Item.Deceleration > 0.0 THEN Dec := Item.Deceleration; ELSE Dec := GVL_1.DATA_RB_B.MOTION_DEC; END_IF;
				IF Item.Jerk > 0.0 THEN Jerk := Item.Jerk; ELSE Jerk := GVL_1.DATA_RB_B.MOTION_JERK; END_IF;
			END_IF
			

            //------------------------------------------------
            // Giá trị dự phòng
            //------------------------------------------------
            IF Vel <= 0.0 THEN
                Vel := 100.0;
            END_IF;

            IF Acc <= 0.0 THEN
                Acc := 1000.0;
            END_IF;

            IF Dec <= 0.0 THEN
                Dec := 1000.0;
            END_IF;

            IF Jerk <= 0.0 THEN
                Jerk := 10000.0;
            END_IF;


            //------------------------------------------------
            // Dynamic Factor
            //------------------------------------------------
            IF AxisGroup.m_id = SCARA_A.m_id THEN
				VelFacLocal    := GVL_1.DATA_RB_A.Fac_Vel;
				AccFacLocal    := GVL_1.DATA_RB_A.Fac_Acc;
				JerkFacLocal   := GVL_1.DATA_RB_A.Fac_Jerk;
				TorqueFacLocal := GVL_1.DATA_RB_A.Fac_Torque;
			ELSE
				VelFacLocal    := GVL_1.DATA_RB_B.Fac_Vel;
				AccFacLocal    := GVL_1.DATA_RB_B.Fac_Acc;
				JerkFacLocal   := GVL_1.DATA_RB_B.Fac_Jerk;
				TorqueFacLocal := GVL_1.DATA_RB_B.Fac_Torque;
			END_IF

            IF VelFacLocal <= 0.0 THEN
                VelFacLocal := 0.1;
            END_IF;

            IF AccFacLocal <= 0.0 THEN
                AccFacLocal := 0.1;
            END_IF;

